KUKA KRL program: MyProgram_142().src

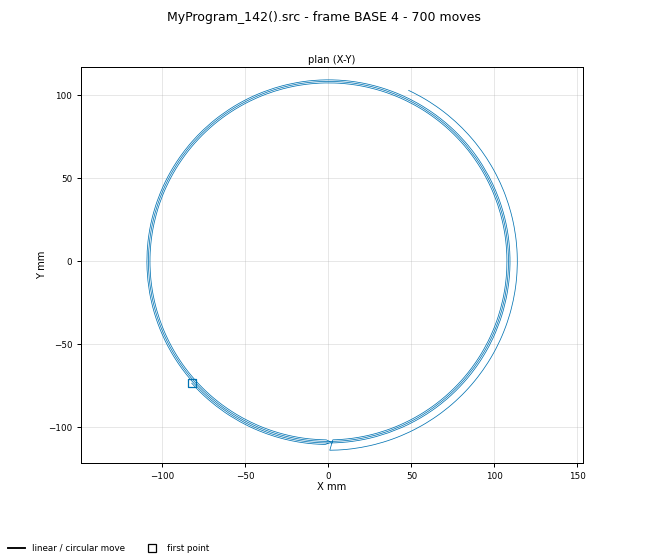
[picture p0: tool path of MyProgram_142().src in frame BASE 4, 700 of 700 moves have a stored position in this frame; points joined in program order, loops and branches not executed]
&ACCESS RVP
&REL 1
&PARAM TEMPLATE = C:\KRC\Roboter\Template\vorgabe
&PARAM EDITMASK = *
DEF MyProgram_142()
; ---- Setting reference (Base) ----
$BASE = BASE_DATA[4]

; --------------------------
; ---- Setting tool (TCP) ----
$TOOL = TOOL_DATA[3]
; --------------------------

$VEL.CP = VEL_APROX_PRINT
Startdeposition()
$VEL.CP = VEL_PRINT
LIN {X -82.3779,Y -73.3835,Z 113,A -141.7997,B 24.948,C -1.666,E1 24.8814,E2 227.604} C_DIS
LIN {X -79.9682,Y -76.004,Z 113,A -139.8537,B 24.948,C -1.6658,E1 24.8851,E2 225.6502} C_DIS
LIN {X -77.4714,Y -78.5454,Z 113,A -138.0878,B 24.9485,C -1.6585,E1 24.8886,E2 223.8941} C_DIS
LIN {X -74.7071,Y -81.1792,Z 113,A -136.1303,B 24.9488,C -1.6534,E1 24.8926,E2 221.9407} C_DIS
LIN {X -72.2466,Y -83.3774,Z 113,A -134.4348,B 24.949,C -1.6493,E1 24.8961,E2 220.2482} C_DIS
LIN {X -67.7785,Y -87.0492,Z 113,A -131.5023,B 24.9496,C -1.6408,E1 24.9025,E2 217.3249} C_DIS
LIN {X -62.2347,Y -91.0947,Z 113,A -127.8013,B 24.9496,C -1.6401,E1 24.9109,E2 213.6125} C_DIS
LIN {X -59.665,Y -92.797,Z 113,A -126.1786,B 24.9496,C -1.6385,E1 24.9147,E2 211.9885} C_DIS
LIN {X -53.2647,Y -96.6148,Z 113,A -122.4009,B 24.9503,C -1.6291,E1 24.9238,E2 208.2219} C_DIS
LIN {X -48.2181,Y -99.2292,Z 113,A -119.3028,B 24.9501,C -1.6312,E1 24.9315,E2 205.1103} C_DIS
LIN {X -45.3422,Y -100.5747,Z 113,A -117.6884,B 24.9503,C -1.628,E1 24.9356,E2 203.4997} C_DIS
LIN {X -41.9036,Y -102.0558,Z 113,A -114.9603,B 24.9485,C -1.6583,E1 24.9428,E2 200.6934} C_DIS
LIN {X -37.221,Y -103.8565,Z 113,A -113.2244,B 24.9508,C -1.6199,E1 24.9472,E2 199.0451} C_DIS
LIN {X -32.1983,Y -105.5211,Z 113,A -110.4618,B 24.9509,C -1.6183,E1 24.9545,E2 196.2811} C_DIS
LIN {X -28.3976,Y -106.6063,Z 113,A -108.4229,B 24.951,C -1.6164,E1 24.96,E2 194.2436} C_DIS
LIN {X -25.5467,Y -107.3263,Z 113,A -106.6947,B 24.9506,C -1.6239,E1 24.9647,E2 192.4952} C_DIS
LIN {X -22.1899,Y -108.0685,Z 113,A -105.0015,B 24.9509,C -1.6193,E1 24.9693,E2 190.8109} C_DIS
LIN {X -18.5186,Y -108.7583,Z 113,A -103.0189,B 24.9508,C -1.6204,E1 24.9748,E2 188.8237} C_DIS
LIN {X -15.3474,Y -109.2505,Z 113,A -101.4417,B 24.9511,C -1.6163,E1 24.9791,E2 187.255} C_DIS
LIN {X -12.6157,Y -109.5996,Z 113,A -100.0275,B 24.9511,C -1.6154,E1 24.983,E2 185.842} C_DIS
LIN {X -9.065,Y -109.9504,Z 113,A -98.0828,B 24.9509,C -1.6191,E1 24.9885,E2 183.8875} C_DIS
LIN {X -5.9741,Y -110.1613,Z 113,A -96.2315,B 24.9503,C -1.6294,E1 24.9937,E2 182.0111} C_DIS
LIN {X -2.0472,Y -110.3041,Z 113,A -94.0279,B 24.9498,C -1.6367,E1 24.9999,E2 179.7901} C_DIS
LIN {X -2.0472,Y -110.3041,Z 113,A -94.0279,B 24.9498,C -1.6367,E1 24.9999,E2 179.7901} C_DIS
Enddeposition()
LIN {X 0.8012,Y -109.3921,Z 113,A -93.8534,B 24.9521,C -1.5983,E1 25.0001,E2 179.7065} C_DIS
Startdeposition()
$VEL.CP = VEL_PRINT
LIN {X -2.7654,Y -109.365,Z 113,A -95.8153,B 24.9524,C -1.594,E1 24.9946,E2 181.6787} C_DIS
LIN {X -5.7929,Y -109.2451,Z 113,A -97.2879,B 24.9521,C -1.5986,E1 24.9905,E2 183.1408} C_DIS
LIN {X -8.9901,Y -109.0286,Z 113,A -98.9104,B 24.952,C -1.6009,E1 24.986,E2 184.7585} C_DIS
LIN {X -12.5666,Y -108.6743,Z 113,A -100.7989,B 24.952,C -1.6009,E1 24.9808,E2 186.6482} C_DIS
LIN {X -15.9909,Y -108.225,Z 113,A -102.74,B 24.9523,C -1.5959,E1 24.9754,E2 188.6028} C_DIS
LIN {X -19.4535,Y -107.6548,Z 113,A -104.4859,B 24.952,C -1.6002,E1 24.9706,E2 190.34} C_DIS
LIN {X -23.1089,Y -106.93,Z 113,A -106.4558,B 24.952,C -1.6003,E1 24.9652,E2 192.312} C_DIS
LIN {X -26.9087,Y -106.0378,Z 113,A -108.7166,B 24.9525,C -1.5927,E1 24.959,E2 194.594} C_DIS
LIN {X -30.6646,Y -105.0138,Z 113,A -110.6107,B 24.952,C -1.5999,E1 24.954,E2 196.4742} C_DIS
LIN {X -34.0937,Y -103.9509,Z 113,A -112.4944,B 24.952,C -1.6012,E1 24.949,E2 198.3582} C_DIS
LIN {X -37.5371,Y -102.7568,Z 113,A -114.8721,B 24.953,C -1.5842,E1 24.9426,E2 200.7808} C_DIS
LIN {X -41.2912,Y -101.3066,Z 113,A -116.4083,B 24.9515,C -1.609,E1 24.9388,E2 202.2615} C_DIS
LIN {X -44.4783,Y -99.9497,Z 113,A -118.2925,B 24.9515,C -1.6082,E1 24.9339,E2 204.1522} C_DIS
LIN {X -47.5492,Y -98.5246,Z 113,A -120.5665,B 24.9526,C -1.5905,E1 24.9281,E2 206.474} C_DIS
LIN {X -51.0831,Y -96.7395,Z 113,A -122.1173,B 24.9512,C -1.6138,E1 24.9244,E2 207.9737} C_DIS
LIN {X -56.8602,Y -93.4607,Z 113,A -125.5555,B 24.9508,C -1.6203,E1 24.9161,E2 211.4066} C_DIS
LIN {X -59.8344,Y -91.5863,Z 113,A -127.5128,B 24.9509,C -1.6186,E1 24.9114,E2 213.3743} C_DIS
LIN {X -66.1199,Y -87.1574,Z 113,A -131.2341,B 24.9498,C -1.6374,E1 24.9031,E2 217.0638} C_DIS
LIN {X -70.5458,Y -83.6155,Z 113,A -134.473,B 24.9501,C -1.6324,E1 24.896,E2 220.3268} C_DIS
LIN {X -73.0132,Y -81.4682,Z 113,A -136.1362,B 24.9497,C -1.6377,E1 24.8925,E2 221.9839} C_DIS
LIN {X -75.4532,Y -79.2163,Z 113,A -138.0378,B 24.9499,C -1.635,E1 24.8886,E2 223.8999} C_DIS
LIN {X -78.1128,Y -76.5934,Z 113,A -139.9944,B 24.9497,C -1.6392,E1 24.8847,E2 225.8547} C_DIS
LIN {X -80.6821,Y -73.881,Z 113,A -141.8513,B 24.9491,C -1.6474,E1 24.8812,E2 227.7003} C_DIS
LIN {X -83.2227,Y -71.0069,Z 113,A -143.8483,B 24.9488,C -1.6524,E1 24.8776,E2 229.6943} C_DIS
LIN {X -85.4937,Y -68.2577,Z 113,A -146.364,B 24.9501,C -1.6322,E1 24.8731,E2 232.27} C_DIS
LIN {X -88.0377,Y -64.9423,Z 113,A -147.7396,B 24.9478,C -1.6685,E1 24.8709,E2 233.5656} C_DIS
LIN {X -90.3611,Y -61.6687,Z 113,A -150.7884,B 24.9497,C -1.6379,E1 24.8659,E2 236.7024} C_DIS
LIN {X -92.8964,Y -57.7779,Z 113,A -152.5487,B 24.9478,C -1.6697,E1 24.8634,E2 238.3959} C_DIS
LIN {X -94.8352,Y -54.537,Z 113,A -154.5071,B 24.9474,C -1.6757,E1 24.8606,E2 240.3501} C_DIS
LIN {X -96.8538,Y -50.866,Z 113,A -156.705,B 24.947,C -1.6816,E1 24.8577,E2 242.5456} C_DIS
LIN {X -98.4649,Y -47.6735,Z 113,A -158.9102,B 24.9475,C -1.6743,E1 24.855,E2 244.78} C_DIS
LIN {X -100.2359,Y -43.8267,Z 113,A -160.6867,B 24.946,C -1.6973,E1 24.853,E2 246.5114} C_DIS
LIN {X -101.4514,Y -40.9354,Z 113,A -162.571,B 24.9463,C -1.693,E1 24.8509,E2 248.4166} C_DIS
LIN {X -102.8244,Y -37.3518,Z 113,A -164.4547,B 24.9456,C -1.7037,E1 24.8491,E2 250.2853} C_DIS
LIN {X -103.9435,Y -34.1167,Z 113,A -166.3425,B 24.9455,C -1.7055,E1 24.8474,E2 252.1797} C_DIS
LIN {X -104.9287,Y -30.9513,Z 113,A -168.2477,B 24.9455,C -1.7044,E1 24.8459,E2 254.0983} C_DIS
LIN {X -105.9399,Y -27.2899,Z 113,A -171.007,B 24.947,C -1.682,E1 24.8439,E2 256.9271} C_DIS
LIN {X -107.201,Y -21.8168,Z 113,A -173.3913,B 24.9451,C -1.7118,E1 24.8426,E2 259.2546} C_DIS
LIN {X -107.798,Y -18.6455,Z 113,A -174.9108,B 24.9443,C -1.7235,E1 24.8419,E2 260.7552} C_DIS
LIN {X -108.7762,Y -11.6534,Z 113,A -178.1709,B 24.9425,C -1.7516,E1 24.8407,E2 263.9678} C_DIS
LIN {X -109.2836,Y -5.0185,Z 113,A 177.3593,B 24.9442,C -1.7262,E1 24.8399,E2 268.5249} C_DIS
LIN {X -109.3981,Y -0.4851,Z 113,A 175.7323,B 24.9418,C -1.7616,E1 24.8398,E2 270.0774} C_DIS
LIN {X -109.2223,Y 6.206,Z 113,A 172.596,B 24.9402,C -1.7867,E1 24.8401,E2 273.1726} C_DIS
LIN {X -108.7527,Y 11.8781,Z 113,A 169.2354,B 24.9405,C -1.7821,E1 24.8408,E2 276.5644} C_DIS
LIN {X -108.4114,Y 14.675,Z 113,A 167.2505,B 24.9414,C -1.768,E1 24.8416,E2 278.5949} C_DIS
LIN {X -107.7858,Y 18.7251,Z 113,A 165.3486,B 24.9404,C -1.7839,E1 24.8424,E2 280.47} C_DIS
LIN {X -107.0836,Y 22.3884,Z 113,A 163.4098,B 24.9399,C -1.7908,E1 24.8435,E2 282.4039} C_DIS
LIN {X -106.2775,Y 25.9441,Z 113,A 161.1299,B 24.9404,C -1.7832,E1 24.845,E2 284.7153} C_DIS
LIN {X -105.3682,Y 29.423,Z 113,A 159.647,B 24.939,C -1.804,E1 24.8461,E2 286.1573} C_DIS
LIN {X -104.0831,Y 33.6853,Z 113,A 157.5878,B 24.9378,C -1.8215,E1 24.8477,E2 288.1865} C_DIS
LIN {X -103.2279,Y 36.2213,Z 113,A 155.9172,B 24.9382,C -1.8158,E1 24.8493,E2 289.8801} C_DIS
LIN {X -101.2858,Y 41.3425,Z 113,A 152.8339,B 24.9382,C -1.8167,E1 24.8524,E2 292.9786} C_DIS
LIN {X -99.7186,Y 44.9911,Z 113,A 150.9412,B 24.9372,C -1.83,E1 24.8545,E2 294.85} C_DIS
LIN {X -98.064,Y 48.4919,Z 113,A 148.8956,B 24.9369,C -1.8354,E1 24.857,E2 296.8937} C_DIS
LIN {X -96.7392,Y 51.0837,Z 113,A 147.4208,B 24.9364,C -1.8418,E1 24.8589,E2 298.3612} C_DIS
LIN {X -95.0536,Y 54.1568,Z 113,A 145.4662,B 24.9364,C -1.8427,E1 24.8616,E2 300.3239} C_DIS
LIN {X -93.3567,Y 57.0314,Z 113,A 143.353,B 24.9369,C -1.8342,E1 24.8647,E2 302.4684} C_DIS
LIN {X -91.542,Y 59.9015,Z 113,A 141.9274,B 24.9357,C -1.8523,E1 24.8668,E2 303.8578} C_DIS
LIN {X -89.57,Y 62.8125,Z 113,A 140.1452,B 24.9352,C -1.8597,E1 24.8696,E2 305.6313} C_DIS
LIN {X -86.8006,Y 66.586,Z 113,A 136.9244,B 24.9367,C -1.8376,E1 24.8751,E2 308.9202} C_DIS
LIN {X -83.8364,Y 70.2828,Z 113,A 135.274,B 24.9341,C -1.8752,E1 24.8779,E2 310.4886} C_DIS
LIN {X -82.098,Y 72.3057,Z 113,A 133.0171,B 24.9361,C -1.8465,E1 24.8822,E2 312.824} C_DIS
LIN {X -78.9179,Y 75.7628,Z 113,A 131.4131,B 24.9334,C -1.8848,E1 24.8851,E2 314.3437} C_DIS
LIN {X -75.4082,Y 79.259,Z 113,A 128.5636,B 24.9336,C -1.8814,E1 24.8909,E2 317.2134} C_DIS
LIN {X -70.6677,Y 83.5117,Z 113,A 125.2283,B 24.9331,C -1.889,E1 24.8978,E2 320.5437} C_DIS
LIN {X -68.3733,Y 85.4021,Z 113,A 123.6376,B 24.933,C -1.8911,E1 24.9013,E2 322.1353} C_DIS
LIN {X -65.5348,Y 87.5969,Z 113,A 121.7948,B 24.9326,C -1.8965,E1 24.9054,E2 323.9719} C_DIS
LIN {X -59.7976,Y 91.6105,Z 113,A 118.3589,B 24.9314,C -1.9127,E1 24.9132,E2 327.381} C_DIS
LIN {X -56.3625,Y 93.7632,Z 113,A 115.9531,B 24.9319,C -1.9058,E1 24.919,E2 329.8108} C_DIS
LIN {X -53.3037,Y 95.5338,Z 113,A 114.2429,B 24.9313,C -1.9145,E1 24.9231,E2 331.5052} C_DIS
LIN {X -50.6765,Y 96.9536,Z 113,A 112.6453,B 24.9312,C -1.9158,E1 24.927,E2 333.1041} C_DIS
LIN {X -48.0598,Y 98.2781,Z 113,A 111.1708,B 24.9308,C -1.9207,E1 24.9307,E2 334.571} C_DIS
LIN {X -45.59,Y 99.4482,Z 113,A 109.2316,B 24.9321,C -1.9032,E1 24.9357,E2 336.5565} C_DIS
LIN {X -42.5907,Y 100.7672,Z 113,A 107.9423,B 24.9307,C -1.9223,E1 24.9389,E2 337.8036} C_DIS
LIN {X -39.2401,Y 102.12,Z 113,A 105.8965,B 24.931,C -1.9189,E1 24.9443,E2 339.8618} C_DIS
LIN {X -32.8544,Y 104.3495,Z 113,A 102.6449,B 24.9298,C -1.9346,E1 24.9528,E2 343.0822} C_DIS
LIN {X -28.269,Y 105.6832,Z 113,A 99.7023,B 24.9309,C -1.9199,E1 24.9608,E2 346.0644} C_DIS
LIN {X -24.7509,Y 106.5617,Z 113,A 97.9468,B 24.9304,C -1.9274,E1 24.9655,E2 347.8046} C_DIS
LIN {X -18.6417,Y 107.8,Z 113,A 94.901,B 24.9295,C -1.9386,E1 24.9738,E2 350.827} C_DIS
LIN {X -15.5709,Y 108.2847,Z 113,A 93.1885,B 24.9297,C -1.9364,E1 24.9786,E2 352.5462} C_DIS
LIN {X -12.4417,Y 108.6889,Z 113,A 91.4662,B 24.9298,C -1.9346,E1 24.9833,E2 354.274} C_DIS
LIN {X -8.7221,Y 109.0501,Z 113,A 89.5604,B 24.9296,C -1.9376,E1 24.9886,E2 356.1736} C_DIS
LIN {X -5.0583,Y 109.2819,Z 113,A 87.5717,B 24.9298,C -1.9357,E1 24.9942,E2 358.1675} C_DIS
LIN {X -1.3425,Y 109.3921,Z 113,A 85.5642,B 24.9298,C -1.9337,E1 24.9998,E2 360.1797} C_DIS
LIN {X 2.3062,Y 109.3744,Z 113,A 83.6652,B 24.9298,C -1.9345,E1 25.0051,E2 362.0767} C_DIS
LIN {X 6.1411,Y 109.2259,Z 113,A 81.768,B 24.9295,C -1.9392,E1 25.0104,E2 363.9623} C_DIS
LIN {X 9.6682,Y 108.9709,Z 113,A 79.8747,B 24.9296,C -1.9374,E1 25.0156,E2 365.8589} C_DIS
LIN {X 13.002,Y 108.6233,Z 113,A 78.0458,B 24.9299,C -1.9341,E1 25.0207,E2 367.6942} C_DIS
LIN {X 16.8027,Y 108.1003,Z 113,A 76.1369,B 24.9296,C -1.9377,E1 25.026,E2 369.5929} C_DIS
LIN {X 20.5395,Y 107.453,Z 113,A 74.1322,B 24.9297,C -1.9361,E1 25.0315,E2 371.599} C_DIS
LIN {X 23.9831,Y 106.7391,Z 113,A 72.0822,B 24.9304,C -1.9267,E1 25.0371,E2 373.6687} C_DIS
LIN {X 27.6095,Y 105.8577,Z 113,A 70.3461,B 24.9298,C -1.9345,E1 25.0418,E2 375.3838} C_DIS
LIN {X 31.3079,Y 104.8229,Z 113,A 68.3615,B 24.9298,C -1.9342,E1 25.0471,E2 377.3658} C_DIS
LIN {X 34.8354,Y 103.7039,Z 113,A 65.8741,B 24.9316,C -1.91,E1 25.0538,E2 379.9057} C_DIS
LIN {X 38.5632,Y 102.3763,Z 113,A 64.6554,B 24.9292,C -1.9433,E1 25.0568,E2 381.0429} C_DIS
LIN {X 41.0421,Y 101.408,Z 113,A 62.9101,B 24.9304,C -1.9273,E1 25.0614,E2 382.8222} C_DIS
LIN {X 44.3336,Y 100.0149,Z 113,A 60.2503,B 24.9329,C -1.8925,E1 25.0684,E2 385.5578} C_DIS
LIN {X 48.9923,Y 97.8159,Z 113,A 58.6274,B 24.9299,C -1.9339,E1 25.0723,E2 387.0785} C_DIS
LIN {X 53.6545,Y 95.3379,Z 113,A 55.7155,B 24.9306,C -1.9239,E1 25.0795,E2 390.0056} C_DIS
LIN {X 56.3723,Y 93.7573,Z 113,A 53.9616,B 24.9311,C -1.9169,E1 25.0837,E2 391.7707} C_DIS
LIN {X 61.0705,Y 90.7656,Z 113,A 50.9637,B 24.9317,C -1.9089,E1 25.0907,E2 394.7777} C_DIS
LIN {X 64.5108,Y 88.3536,Z 113,A 48.6141,B 24.9324,C -1.8988,E1 25.0961,E2 397.143} C_DIS
LIN {X 67.3887,Y 86.1805,Z 113,A 46.9399,B 24.932,C -1.9044,E1 25.0998,E2 398.7978} C_DIS
LIN {X 70.6273,Y 83.5461,Z 113,A 44.7937,B 24.9322,C -1.9019,E1 25.1044,E2 400.9416} C_DIS
LIN {X 73.3173,Y 81.196,Z 113,A 42.8702,B 24.9326,C -1.8959,E1 25.1084,E2 402.8716} C_DIS
LIN {X 75.9181,Y 78.7683,Z 113,A 41.143,B 24.9325,C -1.8979,E1 25.1119,E2 404.5871} C_DIS
LIN {X 78.3464,Y 76.3557,Z 113,A 39.2407,B 24.9331,C -1.8893,E1 25.1156,E2 406.5017} C_DIS
LIN {X 81.9844,Y 72.4358,Z 113,A 36.4618,B 24.9335,C -1.8839,E1 25.1209,E2 409.281} C_DIS
LIN {X 84.1987,Y 69.8468,Z 113,A 33.9749,B 24.9359,C -1.8496,E1 25.1254,E2 411.8374} C_DIS
LIN {X 87.3366,Y 65.8814,Z 113,A 32.1429,B 24.9339,C -1.8782,E1 25.1284,E2 413.5934} C_DIS
LIN {X 89.3104,Y 63.181,Z 113,A 30.4798,B 24.9339,C -1.8776,E1 25.1311,E2 415.2498} C_DIS
LIN {X 90.9002,Y 60.8724,Z 113,A 28.8268,B 24.9347,C -1.8658,E1 25.1337,E2 416.9224} C_DIS
LIN {X 92.8626,Y 57.8322,Z 113,A 27.0985,B 24.9346,C -1.8681,E1 25.1363,E2 418.6366} C_DIS
LIN {X 96.5968,Y 51.3539,Z 113,A 23.357,B 24.9348,C -1.865,E1 25.1415,E2 422.366} C_DIS
LIN {X 98.9562,Y 46.647,Z 113,A 20.5663,B 24.9354,C -1.8557,E1 25.1449,E2 425.1635} C_DIS
LIN {X 100.73,Y 42.6791,Z 113,A 18.1538,B 24.9363,C -1.8432,E1 25.1476,E2 427.5925} C_DIS
LIN {X 102.7796,Y 37.4746,Z 113,A 15.2834,B 24.9367,C -1.8372,E1 25.1505,E2 430.4612} C_DIS
LIN {X 103.9222,Y 34.1824,Z 113,A 13.0549,B 24.9383,C -1.814,E1 25.1525,E2 432.7318} C_DIS
LIN {X 105.387,Y 29.3564,Z 113,A 10.8974,B 24.9374,C -1.8271,E1 25.1542,E2 434.8459} C_DIS
LIN {X 106.1589,Y 26.4299,Z 113,A 9.388,B 24.9375,C -1.8256,E1 25.1552,E2 436.3503} C_DIS
LIN {X 107.0513,Y 22.5459,Z 113,A 7.1063,B 24.9386,C -1.8105,E1 25.1566,E2 438.6544} C_DIS
LIN {X 107.6865,Y 19.2774,Z 113,A 5.4791,B 24.9386,C -1.8102,E1 25.1575,E2 440.2728} C_DIS
LIN {X 108.2497,Y 15.8174,Z 113,A 3.5533,B 24.9392,C -1.8004,E1 25.1583,E2 442.2104} C_DIS
LIN {X 108.6843,Y 12.4812,Z 113,A 1.921,B 24.9392,C -1.8004,E1 25.1589,E2 443.8328} C_DIS
LIN {X 109.0274,Y 9.0051,Z 113,A 0.011,B 24.9399,C -1.791,E1 25.1593,E2 445.7538} C_DIS
LIN {X 109.2436,Y 5.8206,Z 113,A -1.5956,B 24.94,C -1.7885,E1 25.1596,E2 447.3568} C_DIS
LIN {X 109.3762,Y 2.2106,Z 113,A -3.4948,B 24.9405,C -1.7821,E1 25.1598,E2 449.2599} C_DIS
LIN {X 109.3898,Y -1.4676,Z 113,A -5.4893,B 24.9411,C -1.7728,E1 25.1598,E2 451.2644} C_DIS
LIN {X 109.2818,Y -5.0597,Z 113,A -7.3747,B 24.9415,C -1.7665,E1 25.1595,E2 453.1534} C_DIS
LIN {X 108.9967,Y -9.3887,Z 113,A -9.5794,B 24.9418,C -1.7621,E1 25.1591,E2 455.3553} C_DIS
LIN {X 108.6501,Y -12.7727,Z 113,A -11.3391,B 24.9421,C -1.7573,E1 25.1585,E2 457.116} C_DIS
LIN {X 107.9142,Y -17.9587,Z 113,A -14.335,B 24.9434,C -1.7372,E1 25.1573,E2 460.1415} C_DIS
LIN {X 107.1046,Y -22.2864,Z 113,A -16.4,B 24.9432,C -1.7404,E1 25.1562,E2 462.1869} C_DIS
LIN {X 105.4172,Y -29.25,Z 113,A -20.4889,B 24.945,C -1.7136,E1 25.1533,E2 466.3156} C_DIS
LIN {X 104.4469,Y -32.5402,Z 113,A -21.8282,B 24.944,C -1.7281,E1 25.1522,E2 467.6131} C_DIS
LIN {X 103.4702,Y -35.5285,Z 113,A -23.5764,B 24.9447,C -1.7184,E1 25.1507,E2 469.3743} C_DIS
LIN {X 100.7111,Y -42.724,Z 113,A -27.546,B 24.9453,C -1.7088,E1 25.1466,E2 473.3445} C_DIS
LIN {X 99.1808,Y -46.1645,Z 113,A -29.4574,B 24.9455,C -1.7055,E1 25.1444,E2 475.2534} C_DIS
LIN {X 96.7449,Y -51.0728,Z 113,A -32.3463,B 24.9461,C -1.696,E1 25.1408,E2 478.1492} C_DIS
LIN {X 94.812,Y -54.5773,Z 113,A -35.0169,B 24.9481,C -1.6647,E1 25.137,E2 480.8799} C_DIS
LIN {X 92.529,Y -58.3655,Z 113,A -36.5246,B 24.9463,C -1.6934,E1 25.1349,E2 482.312} C_DIS
LIN {X 91.2221,Y -60.3867,Z 113,A -38.4148,B 24.9482,C -1.6623,E1 25.1319,E2 484.2664} C_DIS
LIN {X 89.1168,Y -63.4523,Z 113,A -39.8571,B 24.9472,C -1.679,E1 25.1296,E2 485.6622} C_DIS
LIN {X 86.3725,Y -67.1412,Z 113,A -42.8279,B 24.9491,C -1.6478,E1 25.1245,E2 488.6924} C_DIS
LIN {X 83.791,Y -70.3374,Z 113,A -44.4366,B 24.948,C -1.6658,E1 25.1217,E2 490.2513} C_DIS
LIN {X 81.4672,Y -73.0143,Z 113,A -46.2013,B 24.948,C -1.665,E1 25.1185,E2 492.01} C_DIS
LIN {X 79.0508,Y -75.6249,Z 113,A -48.1269,B 24.9485,C -1.6576,E1 25.1148,E2 493.9447} C_DIS
LIN {X 76.7151,Y -77.9925,Z 113,A -49.8185,B 24.9486,C -1.6555,E1 25.1114,E2 495.6341} C_DIS
LIN {X 73.9902,Y -80.5819,Z 113,A -51.7587,B 24.9489,C -1.652,E1 25.1075,E2 497.5744} C_DIS
LIN {X 71.3802,Y -82.9046,Z 113,A -53.8049,B 24.9497,C -1.6384,E1 25.1031,E2 499.6448} C_DIS
LIN {X 67.4867,Y -86.1016,Z 113,A -56.6817,B 24.9507,C -1.6223,E1 25.0968,E2 502.5488} C_DIS
LIN {X 64.6449,Y -88.2555,Z 113,A -57.9573,B 24.9494,C -1.6439,E1 25.094,E2 503.7688} C_DIS
LIN {X 62.2815,Y -89.9391,Z 113,A -60.1083,B 24.9512,C -1.6136,E1 25.089,E2 505.984} C_DIS
LIN {X 59.1447,Y -92.032,Z 113,A -61.6033,B 24.9502,C -1.6303,E1 25.0856,E2 507.4346} C_DIS
LIN {X 55.4697,Y -94.2929,Z 113,A -63.7913,B 24.9502,C -1.6292,E1 25.0804,E2 509.6185} C_DIS
LIN {X 52.2815,Y -96.0971,Z 113,A -66.5028,B 24.9525,C -1.592,E1 25.0735,E2 512.4101} C_DIS
LIN {X 47.8787,Y -98.3663,Z 113,A -68.1866,B 24.9504,C -1.6264,E1 25.0695,E2 514.008} C_DIS
LIN {X 44.4113,Y -99.9799,Z 113,A -70.5877,B 24.9517,C -1.6063,E1 25.0633,E2 516.4506} C_DIS
LIN {X 36.0671,Y -103.282,Z 113,A -74.9452,B 24.9512,C -1.6144,E1 25.052,E2 520.7795} C_DIS
LIN {X 28.6493,Y -105.5804,Z 113,A -79.1187,B 24.9517,C -1.6051,E1 25.0409,E2 524.9676} C_DIS
LIN {X 24.6705,Y -106.5803,Z 113,A -81.1297,B 24.9515,C -1.6088,E1 25.0354,E2 526.967} C_DIS
LIN {X 21.7324,Y -107.2183,Z 113,A -82.88,B 24.952,C -1.6,E1 25.0306,E2 528.7359} C_DIS
LIN {X 17.9909,Y -107.9089,Z 113,A -84.7608,B 24.9518,C -1.6031,E1 25.0254,E2 530.6072} C_DIS
LIN {X 14.2627,Y -108.4648,Z 113,A -86.7044,B 24.9518,C -1.6031,E1 25.0201,E2 532.5493} C_DIS
LIN {X 11.3431,Y -108.8087,Z 113,A -88.2669,B 24.952,C -1.6012,E1 25.0157,E2 534.1151} C_DIS
LIN {X 6.9829,Y -109.1759,Z 113,A -90.4253,B 24.9517,C -1.6056,E1 25.0097,E2 536.262} C_DIS
LIN {X 4.3324,Y -109.3131,Z 113,A -91.9065,B 24.952,C -1.6013,E1 25.0056,E2 537.7529} C_DIS
LIN {X 1.2624,Y -109.3926,Z 113,A -93.8285,B 24.9528,C -1.5878,E1 25.0001,E2 539.7065} C_DIS
LIN {X 1.2624,Y -109.3926,Z 113,A -93.8285,B 24.9528,C -1.5878,E1 25.0001,E2 539.7065} C_DIS
Enddeposition()
LIN {X 0.8016,Y -108.4705,Z 113,A -93.8436,B 24.9512,C -1.6134,E1 25.0003,E2 539.6609} C_DIS
Startdeposition()
$VEL.CP = VEL_PRINT
LIN {X 4.0415,Y -108.4,Z 113,A -91.1734,B 24.9488,C -1.6536,E1 25.008,E2 536.896} C_DIS
LIN {X 7.9739,Y -108.1818,Z 113,A -89.1291,B 24.9488,C -1.653,E1 25.0137,E2 534.854} C_DIS
LIN {X 11.5542,Y -107.8567,Z 113,A -87.3194,B 24.949,C -1.6503,E1 25.0187,E2 533.0518} C_DIS
LIN {X 15.2018,Y -107.403,Z 113,A -85.3984,B 24.949,C -1.6507,E1 25.024,E2 531.1314} C_DIS
LIN {X 18.8289,Y -106.8275,Z 113,A -83.4484,B 24.9488,C -1.6526,E1 25.0294,E2 529.1789} C_DIS
LIN {X 22.2338,Y -106.1713,Z 113,A -81.5918,B 24.9487,C -1.6553,E1 25.0345,E2 527.3183} C_DIS
LIN {X 28.4242,Y -104.6833,Z 113,A -78.3059,B 24.9487,C -1.6553,E1 25.0434,E2 524.037} C_DIS
LIN {X 34.797,Y -102.7409,Z 113,A -74.7828,B 24.9484,C -1.6597,E1 25.0528,E2 520.5101} C_DIS
LIN {X 37.9726,Y -101.6111,Z 113,A -72.9628,B 24.9481,C -1.6638,E1 25.0575,E2 518.6843} C_DIS
LIN {X 44.0864,Y -99.1119,Z 113,A -69.5353,B 24.948,C -1.6662,E1 25.0664,E2 515.2591} C_DIS
LIN {X 47.3058,Y -97.6155,Z 113,A -67.7699,B 24.948,C -1.6645,E1 25.0708,E2 513.5023} C_DIS
LIN {X 50.6503,Y -95.9222,Z 113,A -65.7577,B 24.9478,C -1.6692,E1 25.0758,E2 511.4845} C_DIS
LIN {X 53.5031,Y -94.3627,Z 113,A -63.8715,B 24.9471,C -1.6795,E1 25.0804,E2 509.5795} C_DIS
LIN {X 56.724,Y -92.4613,Z 113,A -61.8962,B 24.9469,C -1.6832,E1 25.0852,E2 507.6015} C_DIS
LIN {X 60.2765,Y -90.1868,Z 113,A -59.4491,B 24.946,C -1.6972,E1 25.0909,E2 505.1296} C_DIS
LIN {X 63.5812,Y -87.8882,Z 113,A -57.3098,B 24.9457,C -1.7021,E1 25.0958,E2 502.9861} C_DIS
LIN {X 68.1848,Y -84.3645,Z 113,A -54.0748,B 24.9448,C -1.7165,E1 25.1029,E2 499.7292} C_DIS
LIN {X 71.2151,Y -81.8227,Z 113,A -52.5492,B 24.9461,C -1.6965,E1 25.1061,E2 498.2568} C_DIS
LIN {X 73.8298,Y -79.4739,Z 113,A -50.5662,B 24.9454,C -1.7064,E1 25.1102,E2 496.2584} C_DIS
LIN {X 76.4474,Y -76.9571,Z 113,A -48.7093,B 24.9454,C -1.7084,E1 25.1139,E2 494.4045} C_DIS
LIN {X 78.986,Y -74.3486,Z 113,A -46.8645,B 24.9452,C -1.7098,E1 25.1174,E2 492.5644} C_DIS
LIN {X 81.4879,Y -71.5984,Z 113,A -44.8782,B 24.9448,C -1.7158,E1 25.1211,E2 490.5728} C_DIS
LIN {X 83.1038,Y -69.7175,Z 113,A -42.2227,B 24.9407,C -1.7793,E1 25.1261,E2 487.7798} C_DIS
LIN {X 87.7182,Y -63.8133,Z 113,A -39.6834,B 24.9441,C -1.7266,E1 25.1301,E2 485.3769} C_DIS
LIN {X 91.0597,Y -58.9475,Z 113,A -36.268,B 24.9427,C -1.7486,E1 25.1355,E2 481.9266} C_DIS
LIN {X 93.8673,Y -54.3653,Z 113,A -33.7392,B 24.9431,C -1.7431,E1 25.139,E2 479.4238} C_DIS
LIN {X 95.6402,Y -51.1843,Z 113,A -31.7471,B 24.9425,C -1.7518,E1 25.1417,E2 477.4215} C_DIS
LIN {X 97.6494,Y -47.2354,Z 113,A -29.5398,B 24.9425,C -1.7529,E1 25.1444,E2 475.2233} C_DIS
LIN {X 98.7831,Y -44.816,Z 113,A -28.2999,B 24.9426,C -1.7496,E1 25.1459,E2 473.9979} C_DIS
LIN {X 99.938,Y -42.1771,Z 113,A -26.2603,B 24.9408,C -1.7774,E1 25.1482,E2 471.904} C_DIS
LIN {X 101.1465,Y -39.1937,Z 113,A -24.8644,B 24.9413,C -1.7691,E1 25.1496,E2 470.5356} C_DIS
LIN {X 102.3599,Y -35.9019,Z 113,A -23.0977,B 24.9413,C -1.771,E1 25.1512,E2 468.7741} C_DIS
LIN {X 103.4178,Y -32.7362,Z 113,A -21.4254,B 24.9411,C -1.7725,E1 25.1527,E2 467.1077} C_DIS
LIN {X 104.4861,Y -29.1439,Z 113,A -19.3038,B 24.9403,C -1.7852,E1 25.1543,E2 464.9685} C_DIS
LIN {X 105.9416,Y -23.3005,Z 113,A -16.3319,B 24.9403,C -1.786,E1 25.1563,E2 462.0117} C_DIS
LIN {X 106.442,Y -20.899,Z 113,A -13.8196,B 24.9362,C -1.8448,E1 25.1577,E2 459.3755} C_DIS
LIN {X 107.477,Y -14.6811,Z 113,A -11.5165,B 24.9386,C -1.8094,E1 25.1585,E2 457.1695} C_DIS
LIN {X 107.9045,Y -11.0981,Z 113,A -9.7615,B 24.9386,C -1.8089,E1 25.1591,E2 455.4262} C_DIS
LIN {X 108.1829,Y -7.9607,Z 113,A -7.9698,B 24.9379,C -1.82,E1 25.1595,E2 453.6189} C_DIS
LIN {X 108.3918,Y -4.231,Z 113,A -6.004,B 24.9375,C -1.8261,E1 25.1597,E2 451.6503} C_DIS
LIN {X 108.4748,Y -0.1969,Z 113,A -3.8965,B 24.9371,C -1.8319,E1 25.1597,E2 449.5416} C_DIS
LIN {X 108.4184,Y 3.4591,Z 113,A -2.1075,B 24.9371,C -1.8319,E1 25.1597,E2 447.7634} C_DIS
LIN {X 108.24,Y 7.1169,Z 113,A -0.1588,B 24.9366,C -1.8387,E1 25.1594,E2 445.81} C_DIS
LIN {X 107.9555,Y 10.6079,Z 113,A 1.794,B 24.9359,C -1.8492,E1 25.1589,E2 443.8441} C_DIS
LIN {X 107.546,Y 14.1569,Z 113,A 3.5609,B 24.9359,C -1.8499,E1 25.1583,E2 442.086} C_DIS
LIN {X 107.0054,Y 17.7865,Z 113,A 5.5105,B 24.9354,C -1.8566,E1 25.1574,E2 440.1322} C_DIS
LIN {X 106.2965,Y 21.6237,Z 113,A 7.5317,B 24.9351,C -1.8613,E1 25.1563,E2 438.1117} C_DIS
LIN {X 105.5734,Y 24.9203,Z 113,A 9.1919,B 24.9351,C -1.8614,E1 25.1553,E2 436.4608} C_DIS
LIN {X 104.5831,Y 28.7951,Z 113,A 11.2922,B 24.9346,C -1.8674,E1 25.1538,E2 434.3585} C_DIS
LIN {X 103.1854,Y 33.4555,Z 113,A 13.9413,B 24.9338,C -1.8787,E1 25.1517,E2 431.6978} C_DIS
LIN {X 101.9982,Y 36.9182,Z 113,A 15.8722,B 24.9334,C -1.8843,E1 25.1499,E2 429.7645} C_DIS
LIN {X 100.5445,Y 40.7106,Z 113,A 18.0071,B 24.933,C -1.8902,E1 25.1477,E2 427.6276} C_DIS
LIN {X 99.143,Y 44.0175,Z 113,A 19.9124,B 24.9326,C -1.896,E1 25.1455,E2 425.7189} C_DIS
LIN {X 97.8899,Y 46.7349,Z 113,A 21.6723,B 24.9317,C -1.9084,E1 25.1434,E2 423.9392} C_DIS
LIN {X 96.0933,Y 50.3254,Z 113,A 23.5276,B 24.9321,C -1.9027,E1 25.1411,E2 422.1073} C_DIS
LIN {X 94.5124,Y 53.2359,Z 113,A 25.6811,B 24.9305,C -1.9252,E1 25.1381,E2 419.9118} C_DIS
LIN {X 92.8951,Y 56.0102,Z 113,A 27.0233,B 24.9313,C -1.9142,E1 25.1362,E2 418.6026} C_DIS
LIN {X 91.0066,Y 59.0303,Z 113,A 28.8362,B 24.9312,C -1.9162,E1 25.1335,E2 416.7942} C_DIS
LIN {X 88.7412,Y 62.384,Z 113,A 31.3085,B 24.9297,C -1.9362,E1 25.1295,E2 414.2866} C_DIS
LIN {X 83.2478,Y 69.5441,Z 113,A 35.8487,B 24.9296,C -1.9378,E1 25.1217,E2 409.764} C_DIS
LIN {X 80.8479,Y 72.3196,Z 113,A 37.7899,B 24.9293,C -1.9424,E1 25.1181,E2 407.8206} C_DIS
LIN {X 78.1175,Y 75.2606,Z 113,A 39.7514,B 24.9294,C -1.9403,E1 25.1144,E2 405.8727} C_DIS
LIN {X 75.5817,Y 77.808,Z 113,A 41.744,B 24.9288,C -1.9484,E1 25.1104,E2 403.8694} C_DIS
LIN {X 72.753,Y 80.4599,Z 113,A 43.7811,B 24.9286,C -1.9521,E1 25.1062,E2 401.8318} C_DIS
LIN {X 70.1707,Y 82.7202,Z 113,A 45.5669,B 24.9284,C -1.9545,E1 25.1024,E2 400.0472} C_DIS
LIN {X 67.3783,Y 85.0099,Z 113,A 47.4008,B 24.9284,C -1.9549,E1 25.0985,E2 398.2192} C_DIS
LIN {X 63.3687,Y 88.0404,Z 113,A 49.87,B 24.9286,C -1.9517,E1 25.093,E2 395.7665} C_DIS
LIN {X 57.1639,Y 92.1896,Z 113,A 53.9251,B 24.9278,C -1.9628,E1 25.0835,E2 391.6987} C_DIS
LIN {X 54.08,Y 94.0312,Z 113,A 55.8445,B 24.9275,C -1.9665,E1 25.0789,E2 389.7764} C_DIS
LIN {X 50.0566,Y 96.2349,Z 113,A 58.3558,B 24.927,C -1.9735,E1 25.0727,E2 387.2558} C_DIS
LIN {X 46.5453,Y 97.981,Z 113,A 60.6731,B 24.926,C -1.9864,E1 25.0668,E2 384.9139} C_DIS
LIN {X 42.5934,Y 99.7626,Z 113,A 62.7,B 24.9267,C -1.9779,E1 25.0617,E2 382.912} C_DIS
LIN {X 39.497,Y 101.0273,Z 113,A 64.4984,B 24.9264,C -1.981,E1 25.057,E2 381.1103} C_DIS
LIN {X 35.3462,Y 102.555,Z 113,A 66.8432,B 24.9262,C -1.9835,E1 25.0508,E2 378.7645} C_DIS
LIN {X 31.6672,Y 103.7493,Z 113,A 68.8553,B 24.9262,C -1.9838,E1 25.0455,E2 376.7552} C_DIS
LIN {X 29.187,Y 104.4738,Z 113,A 70.2663,B 24.926,C -1.9866,E1 25.0417,E2 375.3399} C_DIS
LIN {X 26.1077,Y 105.2856,Z 113,A 72.2782,B 24.9249,C -2.0013,E1 25.0361,E2 373.2961} C_DIS
LIN {X 22.589,Y 106.0968,Z 113,A 73.8135,B 24.926,C -1.9868,E1 25.032,E2 371.7972} C_DIS
LIN {X 18.7106,Y 106.8488,Z 113,A 75.8653,B 24.926,C -1.9862,E1 25.0264,E2 369.7491} C_DIS
LIN {X 15.2111,Y 107.4017,Z 113,A 77.7532,B 24.926,C -1.9875,E1 25.0212,E2 367.8601} C_DIS
LIN {X 11.4366,Y 107.869,Z 113,A 79.6768,B 24.9262,C -1.9843,E1 25.0159,E2 365.9453} C_DIS
LIN {X 8.3653,Y 108.1508,Z 113,A 81.4003,B 24.9259,C -1.9883,E1 25.0111,E2 364.2134} C_DIS
LIN {X 4.714,Y 108.3711,Z 113,A 83.2079,B 24.9263,C -1.9832,E1 25.0061,E2 362.4185} C_DIS
LIN {X 1.3208,Y 108.4674,Z 113,A 85.1608,B 24.9258,C -1.9894,E1 25.0006,E2 360.4511} C_DIS
LIN {X -2.2772,Y 108.45,Z 113,A 87.0206,B 24.926,C -1.9873,E1 24.9954,E2 358.5961} C_DIS
LIN {X -5.4799,Y 108.3362,Z 113,A 88.6814,B 24.926,C -1.9854,E1 24.9908,E2 356.9394} C_DIS
LIN {X -9.0105,Y 108.0993,Z 113,A 90.5596,B 24.9261,C -1.985,E1 24.9855,E2 355.0616} C_DIS
LIN {X -12.6757,Y 107.7304,Z 113,A 92.4542,B 24.9264,C -1.9819,E1 24.9803,E2 353.1731} C_DIS
LIN {X -16.0723,Y 107.2774,Z 113,A 94.2223,B 24.9266,C -1.979,E1 24.9754,E2 351.4105} C_DIS
LIN {X -19.16,Y 106.768,Z 113,A 96.6333,B 24.9244,C -2.0081,E1 24.9686,E2 348.9277} C_DIS
LIN {X -23.763,Y 105.8407,Z 113,A 98.5354,B 24.9263,C -1.9828,E1 24.9636,E2 347.0836} C_DIS
LIN {X -27.3044,Y 104.9813,Z 113,A 101.1843,B 24.9243,C -2.0098,E1 24.9562,E2 344.3666} C_DIS
LIN {X -32.2607,Y 103.5653,Z 113,A 103.0313,B 24.9271,C -1.9719,E1 24.9515,E2 342.6065} C_DIS
LIN {X -36.7532,Y 102.0583,Z 113,A 105.6198,B 24.9271,C -1.9721,E1 24.9447,E2 340.0125} C_DIS
LIN {X -39.853,Y 100.8875,Z 113,A 107.3861,B 24.9272,C -1.9704,E1 24.9401,E2 338.2466} C_DIS
LIN {X -43.45,Y 99.3912,Z 113,A 109.2935,B 24.9279,C -1.9615,E1 24.9352,E2 336.3558} C_DIS
LIN {X -46.5112,Y 97.9973,Z 113,A 111.1345,B 24.9279,C -1.9613,E1 24.9305,E2 334.5108} C_DIS
LIN {X -49.5708,Y 96.4847,Z 113,A 112.9928,B 24.9279,C -1.9605,E1 24.9259,E2 332.6493} C_DIS
LIN {X -52.8348,Y 94.7364,Z 113,A 114.9937,B 24.9281,C -1.9589,E1 24.921,E2 330.6466} C_DIS
LIN {X -56.2257,Y 92.7642,Z 113,A 117.0128,B 24.9285,C -1.9531,E1 24.9162,E2 328.6353} C_DIS
LIN {X -58.7616,Y 91.1791,Z 113,A 118.6213,B 24.9286,C -1.9512,E1 24.9124,E2 327.0261} C_DIS
LIN {X -62.5413,Y 88.6307,Z 113,A 121.1351,B 24.9286,C -1.9504,E1 24.9066,E2 324.5056} C_DIS
LIN {X -65.3973,Y 86.5436,Z 113,A 123.0045,B 24.929,C -1.9466,E1 24.9024,E2 322.6387} C_DIS
LIN {X -68.355,Y 84.2265,Z 113,A 124.9127,B 24.9295,C -1.9393,E1 24.8982,E2 320.7407} C_DIS
LIN {X -71.019,Y 81.9939,Z 113,A 126.9495,B 24.9292,C -1.9429,E1 24.8939,E2 318.6875} C_DIS
LIN {X -74.2997,Y 79.032,Z 113,A 129.1248,B 24.9301,C -1.9313,E1 24.8895,E2 316.5309} C_DIS
LIN {X -77.441,Y 75.9575,Z 113,A 131.6789,B 24.9298,C -1.9346,E1 24.8844,E2 313.9583} C_DIS
LIN {X -81.1167,Y 72.0193,Z 113,A 134.3397,B 24.9309,C -1.9203,E1 24.8794,E2 311.3196} C_DIS
LIN {X -83.3177,Y 69.46,Z 113,A 136.0766,B 24.9313,C -1.914,E1 24.8763,E2 309.59} C_DIS
LIN {X -85.0367,Y 67.3445,Z 113,A 137.7453,B 24.931,C -1.9188,E1 24.8734,E2 307.9018} C_DIS
LIN {X -87.9279,Y 63.5263,Z 113,A 140.1108,B 24.9319,C -1.9057,E1 24.8695,E2 305.5562} C_DIS
LIN {X -89.8465,Y 60.7792,Z 113,A 141.8152,B 24.9324,C -1.8983,E1 24.8668,E2 303.861} C_DIS
LIN {X -91.646,Y 58.0341,Z 113,A 143.7946,B 24.9321,C -1.9026,E1 24.8638,E2 301.8612} C_DIS
LIN {X -93.9101,Y 54.2907,Z 113,A 145.8232,B 24.9334,C -1.8854,E1 24.8609,E2 299.8634} C_DIS
LIN {X -95.2183,Y 51.9621,Z 113,A 147.4034,B 24.9332,C -1.8876,E1 24.8588,E2 298.2695} C_DIS
LIN {X -96.8798,Y 48.7963,Z 113,A 149.7803,B 24.9323,C -1.9004,E1 24.8557,E2 295.8493} C_DIS
LIN {X -98.5419,Y 45.3457,Z 113,A 151.7807,B 24.9328,C -1.8934,E1 24.8534,E2 293.8547} C_DIS
LIN {X -100.0042,Y 42.0199,Z 113,A 153.802,B 24.9329,C -1.8914,E1 24.8512,E2 291.8268} C_DIS
LIN {X -101.5089,Y 38.2424,Z 113,A 155.4479,B 24.9347,C -1.8658,E1 24.8496,E2 290.2327} C_DIS
LIN {X -102.7681,Y 34.7163,Z 113,A 157.3629,B 24.9353,C -1.8573,E1 24.8479,E2 288.3273} C_DIS
LIN {X -103.8564,Y 31.3143,Z 113,A 159.1848,B 24.9359,C -1.8489,E1 24.8463,E2 286.5148} C_DIS
LIN {X -104.5113,Y 29.0548,Z 113,A 160.6436,B 24.9356,C -1.8531,E1 24.8452,E2 285.0377} C_DIS
LIN {X -105.4242,Y 25.5396,Z 113,A 162.4855,B 24.9363,C -1.8441,E1 24.844,E2 283.2065} C_DIS
LIN {X -106.1277,Y 22.4462,Z 113,A 164.1843,B 24.9366,C -1.8396,E1 24.843,E2 281.5084} C_DIS
LIN {X -106.7509,Y 19.2549,Z 113,A 165.9647,B 24.9368,C -1.8364,E1 24.8421,E2 279.725} C_DIS
LIN {X -107.2629,Y 16.1661,Z 113,A 167.8674,B 24.9365,C -1.8404,E1 24.8413,E2 277.8015} C_DIS
LIN {X -107.7008,Y 12.928,Z 113,A 170.4068,B 24.9348,C -1.8657,E1 24.8404,E2 275.1865} C_DIS
LIN {X -108.2748,Y 6.5903,Z 113,A 173.1207,B 24.9372,C -1.8301,E1 24.8399,E2 272.5412} C_DIS
LIN {X -108.4283,Y 3.1391,Z 113,A 174.7901,B 24.938,C -1.8184,E1 24.8399,E2 270.8897} C_DIS
LIN {X -108.4693,Y -1.067,Z 113,A 176.9646,B 24.9386,C -1.8094,E1 24.8399,E2 268.7236} C_DIS
LIN {X -108.3488,Y -5.2324,Z 113,A 179.8941,B 24.9372,C -1.8298,E1 24.8403,E2 265.7276} C_DIS
LIN {X -107.941,Y -10.749,Z 113,A -178.2396,B 24.9406,C -1.7805,E1 24.8407,E2 263.9678} C_DIS
LIN {X -107.5063,Y -14.4509,Z 113,A -175.8992,B 24.9401,C -1.7882,E1 24.8415,E2 261.5949} C_DIS
LIN {X -106.4275,Y -20.9743,Z 113,A -172.523,B 24.9411,C -1.7728,E1 24.8431,E2 258.2356} C_DIS
LIN {X -105.7707,Y -24.0663,Z 113,A -170.6091,B 24.9408,C -1.7768,E1 24.8443,E2 256.3008} C_DIS
LIN {X -104.6521,Y -28.5398,Z 113,A -168.4022,B 24.9419,C -1.7607,E1 24.8459,E2 254.1195} C_DIS
LIN {X -103.6889,Y -31.8622,Z 113,A -166.8077,B 24.9428,C -1.7464,E1 24.8471,E2 252.55} C_DIS
LIN {X -102.9232,Y -34.2564,Z 113,A -165.1671,B 24.9423,C -1.7542,E1 24.8486,E2 250.8814} C_DIS
LIN {X -101.5457,Y -38.1452,Z 113,A -163.1072,B 24.9431,C -1.7432,E1 24.8505,E2 248.8361} C_DIS
LIN {X -100.5121,Y -40.7901,Z 113,A -161.3769,B 24.9428,C -1.7476,E1 24.8523,E2 247.0856} C_DIS
LIN {X -99.1591,Y -43.9817,Z 113,A -159.3615,B 24.9427,C -1.7493,E1 24.8546,E2 245.0551} C_DIS
LIN {X -97.2611,Y -48.0292,Z 113,A -157.354,B 24.944,C -1.7291,E1 24.857,E2 243.0847} C_DIS
LIN {X -95.5107,Y -51.4231,Z 113,A -155.3182,B 24.9443,C -1.7243,E1 24.8597,E2 241.0497} C_DIS
LIN {X -93.7571,Y -54.557,Z 113,A -153.4133,B 24.9446,C -1.7194,E1 24.8623,E2 239.1464} C_DIS
LIN {X -92.0169,Y -57.4404,Z 113,A -151.3653,B 24.9442,C -1.7251,E1 24.8653,E2 237.0744} C_DIS
LIN {X -89.5413,Y -61.2299,Z 113,A -149.3067,B 24.9454,C -1.7061,E1 24.8685,E2 235.0507} C_DIS
LIN {X -87.6493,Y -63.9073,Z 113,A -147.5082,B 24.9456,C -1.7044,E1 24.8714,E2 233.2476} C_DIS
LIN {X -85.8732,Y -66.2745,Z 113,A -145.6712,B 24.9451,C -1.7111,E1 24.8746,E2 231.3858} C_DIS
LIN {X -82.962,Y -69.8869,Z 113,A -143.3769,B 24.9459,C -1.6993,E1 24.8786,E2 229.1091} C_DIS
LIN {X -80.633,Y -72.5596,Z 113,A -141.5007,B 24.9461,C -1.6952,E1 24.8821,E2 227.2342} C_DIS
LIN {X -78.1243,Y -75.2536,Z 113,A -139.6564,B 24.9467,C -1.687,E1 24.8856,E2 225.4013} C_DIS
LIN {X -75.5932,Y -77.7969,Z 113,A -137.7085,B 24.9467,C -1.685,E1 24.8895,E2 223.45} C_DIS
LIN {X -73.1972,Y -80.0545,Z 113,A -135.9215,B 24.9469,C -1.6834,E1 24.8932,E2 221.6597} C_DIS
LIN {X -70.1455,Y -82.7417,Z 113,A -133.5189,B 24.9465,C -1.6892,E1 24.8983,E2 219.2338} C_DIS
LIN {X -66.2279,Y -85.9091,Z 113,A -131.1481,B 24.9476,C -1.6729,E1 24.9034,E2 216.893} C_DIS
LIN {X -63.2545,Y -88.1219,Z 113,A -128.7769,B 24.9467,C -1.6859,E1 24.9089,E2 214.4827} C_DIS
LIN {X -60.4833,Y -90.0468,Z 113,A -127.2911,B 24.9477,C -1.6712,E1 24.9122,E2 213.0268} C_DIS
LIN {X -57.9021,Y -91.7284,Z 113,A -125.6806,B 24.9479,C -1.668,E1 24.916,E2 211.4188} C_DIS
LIN {X -55.5194,Y -93.1893,Z 113,A -124.0678,B 24.9477,C -1.6713,E1 24.9199,E2 209.7932} C_DIS
LIN {X -51.901,Y -95.2514,Z 113,A -122.0112,B 24.9482,C -1.6625,E1 24.9249,E2 207.7515} C_DIS
LIN {X -48.9589,Y -96.7974,Z 113,A -120.1228,B 24.948,C -1.6656,E1 24.9296,E2 205.8508} C_DIS
LIN {X -45.0288,Y -98.6872,Z 113,A -117.9282,B 24.9485,C -1.6585,E1 24.9352,E2 203.6673} C_DIS
LIN {X -41.8786,Y -100.0638,Z 113,A -116.0882,B 24.9485,C -1.6576,E1 24.9399,E2 201.8254} C_DIS
LIN {X -37.8785,Y -101.6467,Z 113,A -113.8302,B 24.9487,C -1.6548,E1 24.9458,E2 199.5691} C_DIS
LIN {X -34.3132,Y -102.9041,Z 113,A -111.8519,B 24.9488,C -1.6524,E1 24.951,E2 197.5927} C_DIS
LIN {X -30.0147,Y -104.2393,Z 113,A -108.971,B 24.9477,C -1.6713,E1 24.9588,E2 194.6623} C_DIS
LIN {X -26.1735,Y -105.2696,Z 113,A -107.3974,B 24.9491,C -1.6485,E1 24.963,E2 193.1405} C_DIS
LIN {X -23.0995,Y -105.9855,Z 113,A -105.6739,B 24.949,C -1.65,E1 24.9677,E2 191.4111} C_DIS
LIN {X -19.1733,Y -106.7656,Z 113,A -103.6282,B 24.9492,C -1.6464,E1 24.9733,E2 189.3718} C_DIS
LIN {X -15.4202,Y -107.372,Z 113,A -101.6432,B 24.9492,C -1.645,E1 24.9787,E2 187.3886} C_DIS
LIN {X -12.0401,Y -107.8048,Z 113,A -99.786,B 24.9492,C -1.647,E1 24.9839,E2 185.5253} C_DIS
LIN {X -8.9179,Y -108.1067,Z 113,A -98.1374,B 24.9492,C -1.6466,E1 24.9885,E2 183.8768} C_DIS
LIN {X -5.0124,Y -108.3582,Z 113,A -96.2196,B 24.9496,C -1.6405,E1 24.9938,E2 181.9729} C_DIS
LIN {X -2.0343,Y -108.4545,Z 113,A -94.6857,B 24.9496,C -1.6391,E1 24.9981,E2 180.4421} C_DIS
LIN {X 0.8016,Y -108.4705,Z 113,A -93.8414,B 24.9513,C -1.6125,E1 25.0003,E2 179.6609} C_DIS
Enddeposition()
LIN {X 0.8016,Y -108.4705,Z 113,A -93.8414,B 24.9513,C -1.6125,E1 25.0003,E2 179.6609} C_DIS
Startdeposition()
$VEL.CP = VEL_PRINT
LIN {X -1.3239,Y -107.5426,Z 113,A -94.916,B 24.9502,C -1.6309,E1 24.9974,E2 180.692} C_DIS
LIN {X -3.5841,Y -107.4894,Z 113,A -96.1655,B 24.9502,C -1.6289,E1 24.9939,E2 181.9463} C_DIS
LIN {X -6.2176,Y -107.3692,Z 113,A -97.5683,B 24.9502,C -1.6289,E1 24.99,E2 183.3495} C_DIS
LIN {X -8.8457,Y -107.1847,Z 113,A -98.9716,B 24.9502,C -1.6289,E1 24.9861,E2 184.7534} C_DIS
LIN {X -11.4685,Y -106.9358,Z 113,A -100.5263,B 24.9506,C -1.623,E1 24.9817,E2 186.3229} C_DIS
LIN {X -15.1941,Y -106.4701,Z 113,A -102.3754,B 24.9502,C -1.6295,E1 24.9766,E2 188.1582} C_DIS
LIN {X -18.3888,Y -105.967,Z 113,A -104.0582,B 24.9502,C -1.6315,E1 24.972,E2 189.8376} C_DIS
LIN {X -21.8948,Y -105.2968,Z 113,A -105.9622,B 24.9501,C -1.6322,E1 24.9668,E2 191.7421} C_DIS
LIN {X -24.383,Y -104.7484,Z 113,A -107.4014,B 24.9502,C -1.6296,E1 24.9628,E2 193.1892} C_DIS
LIN {X -27.2386,Y -104.0434,Z 113,A -108.876,B 24.95,C -1.6342,E1 24.9589,E2 194.6552} C_DIS
LIN {X -29.9571,Y -103.2944,Z 113,A -110.3935,B 24.95,C -1.6346,E1 24.9548,E2 196.1742} C_DIS
LIN {X -33.3793,Y -102.2381,Z 113,A -112.3475,B 24.95,C -1.6342,E1 24.9496,E2 198.1325} C_DIS
LIN {X -35.8709,Y -101.3907,Z 113,A -113.7521,B 24.9499,C -1.6353,E1 24.9459,E2 199.5373} C_DIS
LIN {X -39.586,Y -99.9988,Z 113,A -115.871,B 24.9498,C -1.6371,E1 24.9403,E2 201.6564} C_DIS
LIN {X -42.3757,Y -98.8507,Z 113,A -117.4388,B 24.9496,C -1.6403,E1 24.9363,E2 203.2202} C_DIS
LIN {X -44.7858,Y -97.7824,Z 113,A -118.8471,B 24.9495,C -1.6417,E1 24.9327,E2 204.6286} C_DIS
LIN {X -46.8284,Y -96.8189,Z 113,A -120.1015,B 24.9495,C -1.6412,E1 24.9295,E2 205.8875} C_DIS
LIN {X -49.5385,Y -95.4625,Z 113,A -121.6684,B 24.9493,C -1.645,E1 24.9257,E2 207.4494} C_DIS
LIN {X -51.5218,Y -94.405,Z 113,A -122.9149,B 24.9493,C -1.6447,E1 24.9226,E2 208.7001} C_DIS
LIN {X -55.298,Y -92.2458,Z 113,A -125.1945,B 24.949,C -1.6495,E1 24.9171,E2 210.9751} C_DIS
LIN {X -58.3293,Y -90.3576,Z 113,A -127.15,B 24.949,C -1.6504,E1 24.9125,E2 212.9347} C_DIS
LIN {X -60.8694,Y -88.6682,Z 113,A -128.7234,B 24.9487,C -1.655,E1 24.9088,E2 214.5024} C_DIS
LIN {X -64.0742,Y -86.3809,Z 113,A -130.8396,B 24.9485,C -1.6579,E1 24.904,E2 216.6191} C_DIS
LIN {X -65.9422,Y -84.9617,Z 113,A -132.1987,B 24.9486,C -1.656,E1 24.901,E2 217.9877} C_DIS
LIN {X -68.7223,Y -82.7283,Z 113,A -134.0508,B 24.9483,C -1.6614,E1 24.897,E2 219.834} C_DIS
LIN {X -71.094,Y -80.7006,Z 113,A -135.8631,B 24.9484,C -1.6589,E1 24.8932,E2 221.6592} C_DIS
LIN {X -73.6854,Y -78.3402,Z 113,A -137.5909,B 24.9479,C -1.668,E1 24.8897,E2 223.3724} C_DIS
LIN {X -75.9156,Y -76.1825,Z 113,A -139.3949,B 24.948,C -1.6658,E1 24.886,E2 225.1894} C_DIS
LIN {X -78.3443,Y -73.6811,Z 113,A -141.1185,B 24.9474,C -1.6749,E1 24.8827,E2 226.8986} C_DIS
LIN {X -80.4374,Y -71.3917,Z 113,A -142.9205,B 24.9476,C -1.673,E1 24.8794,E2 228.7132} C_DIS
LIN {X -82.7083,Y -68.7464,Z 113,A -144.6179,B 24.9469,C -1.6833,E1 24.8763,E2 230.3937} C_DIS
LIN {X -84.3892,Y -66.6723,Z 113,A -146.1169,B 24.9469,C -1.6839,E1 24.8737,E2 231.8985} C_DIS
LIN {X -86.3911,Y -64.0603,Z 113,A -147.793,B 24.9464,C -1.691,E1 24.8709,E2 233.5656} C_DIS
LIN {X -87.9318,Y -61.9287,Z 113,A -149.2063,B 24.9462,C -1.6941,E1 24.8686,E2 234.9786} C_DIS
LIN {X -89.9335,Y -58.981,Z 113,A -151.1063,B 24.9459,C -1.6989,E1 24.8656,E2 236.8765} C_DIS
LIN {X -91.5638,Y -56.4201,Z 113,A -152.742,B 24.9457,C -1.7024,E1 24.8632,E2 238.5121} C_DIS
LIN {X -93.2546,Y -53.5753,Z 113,A -154.5692,B 24.9455,C -1.7048,E1 24.8606,E2 240.3431} C_DIS
LIN {X -94.8548,Y -50.6925,Z 113,A -156.2787,B 24.9451,C -1.7113,E1 24.8583,E2 242.0461} C_DIS
LIN {X -96.4824,Y -47.5178,Z 113,A -158.2366,B 24.9449,C -1.7145,E1 24.8559,E2 244.0068} C_DIS
LIN {X -98.17,Y -43.9257,Z 113,A -160.3206,B 24.9444,C -1.7217,E1 24.8534,E2 246.0852} C_DIS
LIN {X -99.2094,Y -41.5247,Z 113,A -161.7698,B 24.9444,C -1.7237,E1 24.8519,E2 247.5377} C_DIS
LIN {X -100.5352,Y -38.2024,Z 113,A -163.6957,B 24.944,C -1.7285,E1 24.8499,E2 249.4628} C_DIS
LIN {X -101.7018,Y -34.9842,Z 113,A -165.4756,B 24.9435,C -1.7355,E1 24.8482,E2 251.2361} C_DIS
LIN {X -102.5283,Y -32.4826,Z 113,A -166.8911,B 24.9433,C -1.7393,E1 24.847,E2 252.6506} C_DIS
LIN {X -103.2931,Y -29.9614,Z 113,A -168.3026,B 24.943,C -1.7433,E1 24.8459,E2 254.0609} C_DIS
LIN {X -103.9992,Y -27.4103,Z 113,A -169.7234,B 24.9428,C -1.7472,E1 24.8449,E2 255.4805} C_DIS
LIN {X -104.8545,Y -23.9238,Z 113,A -171.6908,B 24.9425,C -1.7512,E1 24.8436,E2 257.45} C_DIS
LIN {X -105.636,Y -20.1935,Z 113,A -173.7373,B 24.9421,C -1.757,E1 24.8425,E2 259.4948} C_DIS
LIN {X -106.1387,Y -17.3624,Z 113,A -175.2891,B 24.9419,C -1.761,E1 24.8417,E2 261.0461} C_DIS
LIN {X -106.5781,Y -14.43,Z 113,A -176.8187,B 24.9414,C -1.7679,E1 24.8411,E2 262.5686} C_DIS
LIN {X -106.9854,Y -10.9957,Z 113,A -178.692,B 24.9411,C -1.7727,E1 24.8405,E2 264.4417} C_DIS
LIN {X -107.2657,Y -7.8182,Z 113,A 179.653,B 24.9406,C -1.7797,E1 24.8402,E2 266.0898} C_DIS
LIN {X -107.4235,Y -5.2232,Z 113,A 178.2385,B 24.9404,C -1.7831,E1 24.8399,E2 267.5047} C_DIS
LIN {X -107.5188,Y -2.6134,Z 113,A 176.8237,B 24.9402,C -1.7867,E1 24.8399,E2 268.9194} C_DIS
LIN {X -107.5499,Y -0.2195,Z 113,A 175.4961,B 24.94,C -1.7889,E1 24.8398,E2 270.2497} C_DIS
LIN {X -107.5188,Y 2.6179,Z 113,A 174.0075,B 24.9396,C -1.7947,E1 24.8398,E2 271.7336} C_DIS
LIN {X -107.4203,Y 5.2942,Z 113,A 172.5756,B 24.9393,C -1.7991,E1 24.84,E2 273.1636} C_DIS
LIN {X -107.2538,Y 7.9815,Z 113,A 171.157,B 24.939,C -1.8043,E1 24.8403,E2 274.5782} C_DIS
LIN {X -107.0297,Y 10.572,Z 113,A 169.7426,B 24.9387,C -1.8078,E1 24.8407,E2 275.9929} C_DIS
LIN {X -106.6364,Y 13.9796,Z 113,A 167.8636,B 24.9385,C -1.8118,E1 24.8413,E2 277.8735} C_DIS
LIN {X -106.2404,Y 16.7273,Z 113,A 166.3528,B 24.9382,C -1.8155,E1 24.8419,E2 279.3846} C_DIS
LIN {X -105.7317,Y 19.6966,Z 113,A 164.7868,B 24.9378,C -1.822,E1 24.8427,E2 280.9442} C_DIS
LIN {X -105.0532,Y 23.0341,Z 113,A 162.8775,B 24.9376,C -1.8244,E1 24.8438,E2 282.8591} C_DIS
LIN {X -104.3297,Y 26.124,Z 113,A 161.2522,B 24.9371,C -1.8322,E1 24.8448,E2 284.4754} C_DIS
LIN {X -103.759,Y 28.2998,Z 113,A 160,B 24.9369,C -1.834,E1 24.8457,E2 285.7304} C_DIS
LIN {X -102.6443,Y 32.1083,Z 113,A 157.9153,B 24.9364,C -1.8418,E1 24.8474,E2 287.8087} C_DIS
LIN {X -101.7007,Y 34.9876,Z 113,A 156.2915,B 24.9361,C -1.8465,E1 24.8488,E2 289.4305} C_DIS
LIN {X -100.8131,Y 37.4683,Z 113,A 154.879,B 24.9358,C -1.8505,E1 24.8502,E2 290.8414} C_DIS
LIN {X -99.9732,Y 39.6512,Z 113,A 153.5737,B 24.9357,C -1.8522,E1 24.8515,E2 292.15} C_DIS
LIN {X -98.8969,Y 42.2661,Z 113,A 152.0943,B 24.9353,C -1.8578,E1 24.8531,E2 293.6243} C_DIS
LIN {X -97.7805,Y 44.7899,Z 113,A 150.6286,B 24.935,C -1.8624,E1 24.8548,E2 295.087} C_DIS
LIN {X -96.0638,Y 48.3621,Z 113,A 148.5032,B 24.9346,C -1.8682,E1 24.8574,E2 297.21} C_DIS
LIN {X -94.8505,Y 50.7006,Z 113,A 147.0902,B 24.9343,C -1.872,E1 24.8592,E2 298.6214} C_DIS
LIN {X -93.3892,Y 53.3411,Z 113,A 145.3841,B 24.9343,C -1.8732,E1 24.8616,E2 300.3339} C_DIS
LIN {X -91.7629,Y 56.0925,Z 113,A 143.7557,B 24.9337,C -1.8808,E1 24.8639,E2 301.9524} C_DIS
LIN {X -90.3526,Y 58.3371,Z 113,A 142.2936,B 24.9335,C -1.883,E1 24.8661,E2 303.4167} C_DIS
LIN {X -88.6833,Y 60.8476,Z 113,A 140.7226,B 24.9331,C -1.8887,E1 24.8685,E2 304.9819} C_DIS
LIN {X -86.3896,Y 64.0625,Z 113,A 138.5893,B 24.9328,C -1.8934,E1 24.872,E2 307.1144} C_DIS
LIN {X -84.4847,Y 66.5515,Z 113,A 136.8745,B 24.9326,C -1.8962,E1 24.875,E2 308.8305} C_DIS
LIN {X -82.7106,Y 68.7436,Z 113,A 135.374,B 24.9323,C -1.9003,E1 24.8776,E2 310.3284} C_DIS
LIN {X -80.6971,Y 71.098,Z 113,A 133.7424,B 24.932,C -1.9052,E1 24.8806,E2 311.9557} C_DIS
LIN {X -78.4545,Y 73.5639,Z 113,A 131.9196,B 24.9318,C -1.9079,E1 24.884,E2 313.78} C_DIS
LIN {X -76.171,Y 75.9273,Z 113,A 130.0236,B 24.9318,C -1.9068,E1 24.8878,E2 315.6867} C_DIS
LIN {X -73.6773,Y 78.3479,Z 113,A 128.3073,B 24.9312,C -1.9163,E1 24.8912,E2 317.3877} C_DIS
LIN {X -71.3922,Y 80.4369,Z 113,A 126.4985,B 24.9313,C -1.9141,E1 24.895,E2 319.2088} C_DIS
LIN {X -68.7256,Y 82.7256,Z 113,A 124.8087,B 24.9305,C -1.9251,E1 24.8985,E2 320.8788} C_DIS
LIN {X -66.6801,Y 84.383,Z 113,A 123.3405,B 24.9305,C -1.9257,E1 24.9018,E2 322.3511} C_DIS
LIN {X -64.068,Y 86.3855,Z 113,A 121.6373,B 24.9301,C -1.9313,E1 24.9055,E2 324.0473} C_DIS
LIN {X -61.9352,Y 87.9271,Z 113,A 120.2309,B 24.9299,C -1.934,E1 24.9087,E2 325.4521} C_DIS
LIN {X -58.9623,Y 89.9459,Z 113,A 118.2632,B 24.9297,C -1.9358,E1 24.9133,E2 327.4221} C_DIS
LIN {X -56.463,Y 91.5371,Z 113,A 116.7199,B 24.9294,C -1.94,E1 24.9169,E2 328.9601} C_DIS
LIN {X -53.3465,Y 93.386,Z 113,A 114.7836,B 24.9292,C -1.9433,E1 24.9216,E2 330.8944} C_DIS
LIN {X -50.707,Y 94.847,Z 113,A 113.1718,B 24.929,C -1.9459,E1 24.9255,E2 332.5047} C_DIS
LIN {X -47.5279,Y 96.4774,Z 113,A 111.2214,B 24.929,C -1.9473,E1 24.9304,E2 334.4571} C_DIS
LIN {X -45.1142,Y 97.6295,Z 113,A 109.8302,B 24.9287,C -1.9507,E1 24.9339,E2 335.8435} C_DIS
LIN {X -42.7101,Y 98.7049,Z 113,A 108.4227,B 24.9285,C -1.9527,E1 24.9375,E2 337.2498} C_DIS
LIN {X -40.2818,Y 99.7205,Z 113,A 106.9734,B 24.9285,C -1.9528,E1 24.9413,E2 338.7019} C_DIS
LIN {X -37.4717,Y 100.8119,Z 113,A 105.4054,B 24.9282,C -1.9564,E1 24.9453,E2 340.2647} C_DIS
LIN {X -34.9714,Y 101.7062,Z 113,A 103.9948,B 24.9281,C -1.9583,E1 24.949,E2 341.6734} C_DIS
LIN {X -32.4974,Y 102.5235,Z 113,A 102.5701,B 24.9281,C -1.9586,E1 24.9528,E2 343.1002} C_DIS
LIN {X -29.9165,Y 103.3059,Z 113,A 101.1742,B 24.9278,C -1.9617,E1 24.9566,E2 344.4909} C_DIS
LIN {X -27.393,Y 104.0037,Z 113,A 99.7657,B 24.9278,C -1.9627,E1 24.9604,E2 345.8994} C_DIS
LIN {X -23.9449,Y 104.8496,Z 113,A 97.6804,B 24.9282,C -1.957,E1 24.9661,E2 348.001} C_DIS
LIN {X -20.3445,Y 105.607,Z 113,A 95.8384,B 24.9277,C -1.9632,E1 24.9711,E2 349.8303} C_DIS
LIN {X -17.4616,Y 106.1221,Z 113,A 94.1487,B 24.928,C -1.9593,E1 24.9758,E2 351.5309} C_DIS
LIN {X -13.8627,Y 106.6516,Z 113,A 92.3251,B 24.9276,C -1.965,E1 24.9808,E2 353.3424} C_DIS
LIN {X -10.5329,Y 107.0337,Z 113,A 90.6107,B 24.9273,C -1.9687,E1 24.9855,E2 355.0491} C_DIS
LIN {X -7.9076,Y 107.2596,Z 113,A 89.2035,B 24.9273,C -1.9692,E1 24.9894,E2 356.4557} C_DIS
LIN {X -5.2789,Y 107.4211,Z 113,A 87.797,B 24.9273,C -1.9696,E1 24.9933,E2 357.8617} C_DIS
LIN {X -2.0702,Y 107.5288,Z 113,A 86.0214,B 24.9274,C -1.9675,E1 24.9983,E2 359.6424} C_DIS
LIN {X 1.3283,Y 107.5425,Z 113,A 84.2756,B 24.9272,C -1.9704,E1 25.0032,E2 361.3812} C_DIS
LIN {X 3.5798,Y 107.4895,Z 113,A 83.0327,B 24.9273,C -1.9688,E1 25.0066,E2 362.6276} C_DIS
LIN {X 6.2117,Y 107.3696,Z 113,A 81.6287,B 24.9273,C -1.9688,E1 25.0106,E2 364.0311} C_DIS
LIN {X 9.8445,Y 107.0972,Z 113,A 79.6845,B 24.9273,C -1.9686,E1 25.016,E2 365.9749} C_DIS
LIN {X 13.1728,Y 106.741,Z 113,A 77.9498,B 24.9273,C -1.9702,E1 25.0208,E2 367.7045} C_DIS
LIN {X 16.7074,Y 106.2435,Z 113,A 76.0052,B 24.9273,C -1.968,E1 25.0261,E2 369.6527} C_DIS
LIN {X 19.6811,Y 105.7346,Z 113,A 74.4417,B 24.9273,C -1.9691,E1 25.0304,E2 371.2117} C_DIS
LIN {X 23.2243,Y 105.0117,Z 113,A 72.472,B 24.9275,C -1.9665,E1 25.0358,E2 373.1852} C_DIS
LIN {X 26.141,Y 104.3255,Z 113,A 70.926,B 24.9275,C -1.9676,E1 25.04,E2 374.7264} C_DIS
LIN {X 28.3291,Y 103.751,Z 113,A 69.6751,B 24.9276,C -1.965,E1 25.0434,E2 375.9815} C_DIS
LIN {X 32.1172,Y 102.6416,Z 113,A 67.6194,B 24.9276,C -1.9653,E1 25.0489,E2 378.0328} C_DIS
LIN {X 34.9811,Y 101.7029,Z 113,A 66.0174,B 24.9276,C -1.9641,E1 25.0531,E2 379.6346} C_DIS
LIN {X 37.4791,Y 100.8091,Z 113,A 64.6087,B 24.9278,C -1.963,E1 25.0568,E2 381.0429} C_DIS
LIN {X 41.1586,Y 99.3636,Z 113,A 62.5045,B 24.9279,C -1.9609,E1 25.0623,E2 383.1473} C_DIS
LIN {X 43.9577,Y 98.1555,Z 113,A 60.789,B 24.9283,C -1.9554,E1 25.0667,E2 384.8718} C_DIS
LIN {X 46.8372,Y 96.8147,Z 113,A 59.1962,B 24.9282,C -1.9574,E1 25.0707,E2 386.4557} C_DIS
LIN {X 49.527,Y 95.4685,Z 113,A 57.5986,B 24.9283,C -1.9555,E1 25.0747,E2 388.0534} C_DIS
LIN {X 51.5307,Y 94.4002,Z 113,A 56.3491,B 24.9285,C -1.9522,E1 25.0777,E2 389.307} C_DIS
LIN {X 54.1588,Y 92.9192,Z 113,A 54.7909,B 24.9285,C -1.9519,E1 25.0815,E2 390.8613} C_DIS
LIN {X 57.2925,Y 91.0189,Z 113,A 52.8463,B 24.9288,C -1.9493,E1 25.0861,E2 392.8059} C_DIS
LIN {X 59.7859,Y 89.4022,Z 113,A 51.2732,B 24.9289,C -1.9471,E1 25.0898,E2 394.379} C_DIS
LIN {X 62.6933,Y 87.3863,Z 113,A 49.348,B 24.9293,C -1.9423,E1 25.0942,E2 396.3091} C_DIS
LIN {X 65.6475,Y 85.1888,Z 113,A 47.394,B 24.9295,C -1.9391,E1 25.0986,E2 398.2636} C_DIS
LIN {X 68.078,Y 83.2606,Z 113,A 45.6908,B 24.9299,C -1.9338,E1 25.1023,E2 399.9727} C_DIS
LIN {X 70.7388,Y 81.0108,Z 113,A 43.8945,B 24.9299,C -1.9327,E1 25.1061,E2 401.7646} C_DIS
LIN {X 73.0632,Y 78.9222,Z 113,A 42.2819,B 24.9301,C -1.9315,E1 25.1094,E2 403.3735} C_DIS
LIN {X 75.4444,Y 76.6479,Z 113,A 40.4838,B 24.9305,C -1.926,E1 25.113,E2 405.1772} C_DIS
LIN {X 77.5648,Y 74.5015,Z 113,A 38.876,B 24.9307,C -1.9225,E1 25.1162,E2 406.7864} C_DIS
LIN {X 79.9943,Y 71.8866,Z 113,A 36.9875,B 24.931,C -1.9187,E1 25.1197,E2 408.6754} C_DIS
LIN {X 81.9934,Y 69.5978,Z 113,A 35.3867,B 24.9312,C -1.9157,E1 25.1226,E2 410.276} C_DIS
LIN {X 84.2795,Y 66.8111,Z 113,A 33.4752,B 24.9315,C -1.9115,E1 25.126,E2 412.1886} C_DIS
LIN {X 86.1846,Y 64.3355,Z 113,A 31.8738,B 24.9316,C -1.9101,E1 25.1287,E2 413.7858} C_DIS
LIN {X 87.9361,Y 61.9225,Z 113,A 30.2878,B 24.9319,C -1.9062,E1 25.1313,E2 415.3733} C_DIS
LIN {X 89.9412,Y 58.9694,Z 113,A 28.3541,B 24.9323,C -1.8999,E1 25.1343,E2 417.3122} C_DIS
LIN {X 92.2478,Y 55.2947,Z 113,A 26.0976,B 24.9326,C -1.8961,E1 25.1376,E2 419.5662} C_DIS
LIN {X 93.3975,Y 53.3266,Z 113,A 24.8909,B 24.9328,C -1.8932,E1 25.1393,E2 420.7735} C_DIS
LIN {X 94.8533,Y 50.6953,Z 113,A 23.2995,B 24.9331,C -1.8892,E1 25.1414,E2 422.366} C_DIS
LIN {X 96.4771,Y 47.5287,Z 113,A 21.3675,B 24.9336,C -1.8824,E1 25.1439,E2 424.3039} C_DIS
LIN {X 98.1662,Y 43.9341,Z 113,A 19.3102,B 24.9338,C -1.8788,E1 25.1463,E2 426.3584} C_DIS
LIN {X 99.2129,Y 41.5164,Z 113,A 17.9259,B 24.9341,C -1.8756,E1 25.1478,E2 427.7427} C_DIS
LIN {X 100.3491,Y 38.6938,Z 113,A 16.3065,B 24.9344,C -1.8709,E1 25.1495,E2 429.3644} C_DIS
LIN {X 101.1047,Y 36.6689,Z 113,A 15.101,B 24.9348,C -1.8651,E1 25.1506,E2 430.5766} C_DIS
LIN {X 101.9998,Y 34.1004,Z 113,A 13.7047,B 24.9349,C -1.8631,E1 25.1519,E2 431.9699} C_DIS
LIN {X 102.9261,Y 31.1988,Z 113,A 12.1142,B 24.9352,C -1.8595,E1 25.1532,E2 433.5598} C_DIS
LIN {X 103.551,Y 29.0515,Z 113,A 10.8848,B 24.9355,C -1.8542,E1 25.1541,E2 434.7945} C_DIS
LIN {X 104.5415,Y 25.2558,Z 113,A 8.8449,B 24.9358,C -1.8499,E1 25.1556,E2 436.8329} C_DIS
LIN {X 105.1067,Y 22.7889,Z 113,A 7.435,B 24.9363,C -1.8431,E1 25.1564,E2 438.2507} C_DIS
LIN {X 105.7342,Y 19.6837,Z 113,A 5.8344,B 24.9364,C -1.8415,E1 25.1573,E2 439.8456} C_DIS
LIN {X 106.3859,Y 15.786,Z 113,A 3.7424,B 24.9369,C -1.8354,E1 25.1582,E2 441.9398} C_DIS
LIN {X 106.7753,Y 12.88,Z 113,A 2.0812,B 24.9375,C -1.8261,E1 25.1588,E2 443.613} C_DIS
LIN {X 107.1192,Y 9.6065,Z 113,A 0.4084,B 24.9376,C -1.824,E1 25.1592,E2 445.2809} C_DIS
LIN {X 107.3224,Y 6.9798,Z 113,A -0.9859,B 24.9379,C -1.8199,E1 25.1595,E2 446.6767} C_DIS
LIN {X 107.4611,Y 4.3489,Z 113,A -2.4989,B 24.9386,C -1.8106,E1 25.1597,E2 448.2025} C_DIS
LIN {X 107.548,Y 0.5646,Z 113,A -4.4441,B 24.9388,C -1.8072,E1 25.1597,E2 450.1443} C_DIS
LIN {X 107.5183,Y -2.6411,Z 113,A -6.0366,B 24.9388,C -1.8066,E1 25.1597,E2 451.7286} C_DIS
LIN {X 107.4297,Y -5.0788,Z 113,A -7.3111,B 24.939,C -1.8035,E1 25.1596,E2 453.0029} C_DIS
LIN {X 107.2599,Y -7.9035,Z 113,A -8.8227,B 24.9394,C -1.7984,E1 25.1593,E2 454.5175} C_DIS
LIN {X 107.0325,Y -10.5451,Z 113,A -10.2253,B 24.9397,C -1.7942,E1 25.1589,E2 455.9217} C_DIS
LIN {X 106.6215,Y -14.0951,Z 113,A -12.1762,B 24.9402,C -1.786,E1 25.1583,E2 457.8804} C_DIS
LIN {X 106.1807,Y -17.1111,Z 113,A -13.9037,B 24.9409,C -1.7762,E1 25.1575,E2 459.6208} C_DIS
LIN {X 105.5428,Y -20.6776,Z 113,A -15.6157,B 24.9406,C -1.7795,E1 25.1567,E2 461.3151} C_DIS
LIN {X 105.0212,Y -23.181,Z 113,A -17.0596,B 24.9412,C -1.7716,E1 25.1558,E2 462.7693} C_DIS
LIN {X 104.3214,Y -26.1567,Z 113,A -18.6118,B 24.9413,C -1.7697,E1 25.1548,E2 464.3171} C_DIS
LIN {X 103.753,Y -28.3216,Z 113,A -19.823,B 24.9416,C -1.7651,E1 25.1539,E2 465.5321} C_DIS
LIN {X 103.0234,Y -30.8707,Z 113,A -21.2036,B 24.9418,C -1.762,E1 25.1528,E2 466.9121} C_DIS
LIN {X 102.2381,Y -33.3792,Z 113,A -22.5619,B 24.942,C -1.7594,E1 25.1517,E2 468.2689} C_DIS
LIN {X 101.3917,Y -35.8683,Z 113,A -24.0278,B 24.9425,C -1.7521,E1 25.1503,E2 469.7435} C_DIS
LIN {X 100.0087,Y -39.5608,Z 113,A -26.1162,B 24.9429,C -1.7461,E1 25.1482,E2 471.8344} C_DIS
LIN {X 98.8511,Y -42.3749,Z 113,A -27.8261,B 24.9434,C -1.7373,E1 25.1464,E2 473.5559} C_DIS
LIN {X 97.491,Y -45.4118,Z 113,A -29.493,B 24.9434,C -1.7365,E1 25.1445,E2 475.2156} C_DIS
LIN {X 96.0598,Y -48.3701,Z 113,A -31.1821,B 24.9437,C -1.7338,E1 25.1424,E2 476.9019} C_DIS
LIN {X 94.8475,Y -50.7061,Z 113,A -32.5732,B 24.9439,C -1.7301,E1 25.1406,E2 478.2944} C_DIS
LIN {X 93.5782,Y -53.012,Z 113,A -34.153,B 24.9447,C -1.7183,E1 25.1384,E2 479.8938} C_DIS
LIN {X 91.71,Y -56.1797,Z 113,A -35.9149,B 24.9445,C -1.7212,E1 25.1359,E2 481.6399} C_DIS
LIN {X 90.3286,Y -58.3746,Z 113,A -37.3376,B 24.9448,C -1.7155,E1 25.1337,E2 483.069} C_DIS
LIN {X 88.6735,Y -60.8618,Z 113,A -38.8629,B 24.945,C -1.7138,E1 25.1313,E2 484.5906} C_DIS
LIN {X 86.3953,Y -64.0547,Z 113,A -40.9467,B 24.9453,C -1.7083,E1 25.1279,E2 486.6773} C_DIS
LIN {X 84.2884,Y -66.7998,Z 113,A -42.8448,B 24.9458,C -1.701,E1 25.1247,E2 488.5837} C_DIS
LIN {X 81.9915,Y -69.6,Z 113,A -44.7532,B 24.946,C -1.6968,E1 25.1213,E2 490.4932} C_DIS
LIN {X 80.1057,Y -71.7621,Z 113,A -46.2969,B 24.9463,C -1.6922,E1 25.1184,E2 492.0409} C_DIS
LIN {X 78.0199,Y -74.026,Z 113,A -48.0343,B 24.9469,C -1.6839,E1 25.1151,E2 493.7904} C_DIS
LIN {X 75.5801,Y -76.5139,Z 113,A -49.7391,B 24.9467,C -1.6858,E1 25.1117,E2 495.4833} C_DIS
LIN {X 73.2034,Y -78.7935,Z 113,A -51.5623,B 24.9472,C -1.6787,E1 25.108,E2 497.316} C_DIS
LIN {X 70.5715,Y -81.157,Z 113,A -53.3374,B 24.9472,C -1.679,E1 25.1043,E2 499.0832} C_DIS
LIN {X 68.0036,Y -83.3209,Z 113,A -55.2214,B 24.9477,C -1.6709,E1 25.1002,E2 500.9791} C_DIS
LIN {X 65.2434,Y -85.5002,Z 113,A -56.9822,B 24.9477,C -1.6716,E1 25.0964,E2 502.7318} C_DIS
LIN {X 63.3042,Y -86.9447,Z 113,A -58.2862,B 24.9478,C -1.6682,E1 25.0934,E2 504.0391} C_DIS
LIN {X 60.8212,Y -88.7012,Z 113,A -59.8466,B 24.9478,C -1.6674,E1 25.0899,E2 505.596} C_DIS
LIN {X 57.5254,Y -90.8734,Z 113,A -61.9523,B 24.9482,C -1.6632,E1 25.0849,E2 507.7048} C_DIS
LIN {X 55.2854,Y -92.2533,Z 113,A -63.3465,B 24.9483,C -1.6609,E1 25.0816,E2 509.1002} C_DIS
LIN {X 52.1966,Y -94.0336,Z 113,A -65.284,B 24.9486,C -1.6559,E1 25.0769,E2 511.0438} C_DIS
LIN {X 48.9881,Y -95.7439,Z 113,A -67.2415,B 24.9489,C -1.6517,E1 25.072,E2 513.0056} C_DIS
LIN {X 45.9817,Y -97.2257,Z 113,A -68.9504,B 24.9489,C -1.652,E1 25.0677,E2 514.7093} C_DIS
LIN {X 42.683,Y -98.7167,Z 113,A -70.8734,B 24.949,C -1.6493,E1 25.0628,E2 516.634} C_DIS
LIN {X 40.2605,Y -99.7292,Z 113,A -72.2818,B 24.9492,C -1.6468,E1 25.0592,E2 518.0449} C_DIS
LIN {X 37.4592,Y -100.8164,Z 113,A -73.8576,B 24.9492,C -1.6457,E1 25.0551,E2 519.62} C_DIS
LIN {X 34.9865,Y -101.7011,Z 113,A -75.2591,B 24.9494,C -1.6438,E1 25.0514,E2 521.0232} C_DIS
LIN {X 32.423,Y -102.5468,Z 113,A -76.6835,B 24.9494,C -1.6426,E1 25.0476,E2 522.4477} C_DIS
LIN {X 29.9368,Y -103.3002,Z 113,A -78.0653,B 24.9495,C -1.6411,E1 25.0439,E2 523.8307} C_DIS
LIN {X 27.429,Y -103.9942,Z 113,A -79.4537,B 24.9496,C -1.6395,E1 25.0402,E2 525.2206} C_DIS
LIN {X 24.0163,Y -104.8331,Z 113,A -81.3693,B 24.9499,C -1.6359,E1 25.0349,E2 527.142} C_DIS
LIN {X 20.9684,Y -105.4868,Z 113,A -82.9819,B 24.9499,C -1.6364,E1 25.0305,E2 528.7514} C_DIS
LIN {X 17.4566,Y -106.1229,Z 113,A -84.9237,B 24.95,C -1.6332,E1 25.0252,E2 530.6985} C_DIS
LIN {X 14.4735,Y -106.5724,Z 113,A -86.4859,B 24.95,C -1.6339,E1 25.0209,E2 532.2578} C_DIS
LIN {X 11.1806,Y -106.966,Z 113,A -88.3024,B 24.9502,C -1.6309,E1 25.0158,E2 534.0802} C_DIS
LIN {X 8.0834,Y -107.2456,Z 113,A -89.8906,B 24.95,C -1.6328,E1 25.0114,E2 535.6629} C_DIS
LIN {X 5.2717,Y -107.4214,Z 113,A -91.4027,B 24.9501,C -1.6317,E1 25.0072,E2 537.177} C_DIS
LIN {X 2.6394,Y -107.5184,Z 113,A -92.8076,B 24.9501,C -1.6312,E1 25.0033,E2 538.5829} C_DIS
LIN {X 2.6394,Y -107.5184,Z 113,A -92.8076,B 24.9501,C -1.6312,E1 25.0033,E2 538.5829} C_DIS
Enddeposition()
LIN {X 0.7991,Y -113.7938,Z 114,A -93.153,B 24.9546,C -1.5563,E1 25.0018,E2 539.1057} C_DIS
Startdeposition()
$VEL.CP = VEL_PRINT
LIN {X 3.1462,Y -113.7549,Z 114,A -91.7689,B 24.9541,C -1.5655,E1 25.0057,E2 537.7001} C_DIS
LIN {X 5.5839,Y -113.663,Z 114,A -90.4389,B 24.9538,C -1.5704,E1 25.0095,E2 536.3589} C_DIS
LIN {X 8.7285,Y -113.4632,Z 114,A -88.9583,B 24.954,C -1.5665,E1 25.0136,E2 534.8882} C_DIS
LIN {X 11.5104,Y -113.2148,Z 114,A -87.6952,B 24.9543,C -1.561,E1 25.017,E2 533.639} C_DIS
LIN {X 14.2853,Y -112.8982,Z 114,A -86.149,B 24.9539,C -1.568,E1 25.0214,E2 532.0773} C_DIS
LIN {X 17.0517,Y -112.5136,Z 114,A -84.7451,B 24.9539,C -1.5689,E1 25.0253,E2 530.6726} C_DIS
LIN {X 19.4555,Y -112.1246,Z 114,A -83.521,B 24.9539,C -1.5697,E1 25.0286,E2 529.4478} C_DIS
LIN {X 22.5519,Y -111.5414,Z 114,A -82.1006,B 24.9542,C -1.5637,E1 25.0325,E2 528.0433} C_DIS
LIN {X 24.9337,Y -111.0349,Z 114,A -80.7139,B 24.9537,C -1.572,E1 25.0363,E2 526.6388} C_DIS
LIN {X 27.9979,Y -110.3005,Z 114,A -79.1309,B 24.9537,C -1.5734,E1 25.0406,E2 525.0547} C_DIS
LIN {X 30.6963,Y -109.5802,Z 114,A -77.7279,B 24.9535,C -1.5748,E1 25.0444,E2 523.6508} C_DIS
LIN {X 33.0344,Y -108.8999,Z 114,A -76.5049,B 24.9535,C -1.576,E1 25.0477,E2 522.4269} C_DIS
LIN {X 35.697,Y -108.0564,Z 114,A -75.1024,B 24.9534,C -1.5776,E1 25.0514,E2 521.0234} C_DIS
LIN {X 38.3381,Y -107.1478,Z 114,A -73.6999,B 24.9533,C -1.5793,E1 25.0551,E2 519.6197} C_DIS
LIN {X 41.2893,Y -106.0437,Z 114,A -72.1183,B 24.9532,C -1.5812,E1 25.0592,E2 518.0369} C_DIS
LIN {X 43.8793,Y -104.9985,Z 114,A -70.7163,B 24.953,C -1.5831,E1 25.0628,E2 516.6337} C_DIS
LIN {X 46.4428,Y -103.89,Z 114,A -69.3146,B 24.953,C -1.585,E1 25.0664,E2 515.2308} C_DIS
LIN {X 48.6558,Y -102.874,Z 114,A -67.9632,B 24.9525,C -1.5926,E1 25.0699,E2 513.865} C_DIS
LIN {X 51.4845,Y -101.4861,Z 114,A -66.512,B 24.9527,C -1.5892,E1 25.0735,E2 512.4259} C_DIS
LIN {X 53.9596,Y -100.192,Z 114,A -65.1108,B 24.9525,C -1.5914,E1 25.0769,E2 511.0234} C_DIS
LIN {X 56.0918,Y -99.0159,Z 114,A -63.8895,B 24.9525,C -1.5933,E1 25.0799,E2 509.8012} C_DIS
LIN {X 58.8108,Y -97.4236,Z 114,A -62.3094,B 24.9523,C -1.596,E1 25.0837,E2 508.2196} C_DIS
LIN {X 61.184,Y -95.951,Z 114,A -61.072,B 24.9526,C -1.591,E1 25.0866,E2 506.9979} C_DIS
LIN {X 63.2239,Y -94.6213,Z 114,A -59.5586,B 24.9516,C -1.6066,E1 25.0902,E2 505.4528} C_DIS
LIN {X 65.8184,Y -92.8333,Z 114,A -58.2713,B 24.9523,C -1.5961,E1 25.0931,E2 504.1945} C_DIS
LIN {X 68.0768,Y -91.19,Z 114,A -56.8713,B 24.9521,C -1.5988,E1 25.0962,E2 502.7932} C_DIS
LIN {X 70.2942,Y -89.4919,Z 114,A -55.4715,B 24.9519,C -1.6016,E1 25.0993,E2 501.392} C_DIS
LIN {X 72.194,Y -87.9686,Z 114,A -53.9595,B 24.951,C -1.6174,E1 25.1027,E2 499.8483} C_DIS
LIN {X 74.3311,Y -86.1704,Z 114,A -52.56,B 24.9508,C -1.6203,E1 25.1056,E2 498.4475} C_DIS
LIN {X 76.6872,Y -84.0782,Z 114,A -51.111,B 24.951,C -1.6177,E1 25.1086,E2 497.0104} C_DIS
LIN {X 78.7275,Y -82.1709,Z 114,A -49.7118,B 24.9508,C -1.6208,E1 25.1115,E2 495.6097} C_DIS
LIN {X 80.4688,Y -80.4688,Z 114,A -48.492,B 24.9506,C -1.6235,E1 25.1139,E2 494.3887} C_DIS
LIN {X 82.4194,Y -78.4697,Z 114,A -47.0935,B 24.9504,C -1.6266,E1 25.1166,E2 492.9887} C_DIS
LIN {X 84.3203,Y -76.4234,Z 114,A -45.5656,B 24.9499,C -1.6359,E1 25.1195,E2 491.4459} C_DIS
LIN {X 86.1704,Y -74.3311,Z 114,A -44.161,B 24.9496,C -1.6395,E1 25.1221,E2 490.0392} C_DIS
LIN {X 88.194,Y -71.9159,Z 114,A -42.8814,B 24.9502,C -1.6295,E1 25.1243,E2 488.7891} C_DIS
LIN {X 89.9324,Y -69.7298,Z 114,A -41.4834,B 24.95,C -1.6329,E1 25.1267,E2 487.3895} C_DIS
LIN {X 91.6165,Y -67.5018,Z 114,A -40.0853,B 24.9498,C -1.6363,E1 25.1291,E2 485.99} C_DIS
LIN {X 93.0412,Y -65.527,Z 114,A -38.5748,B 24.9488,C -1.6529,E1 25.1316,E2 484.4476} C_DIS
LIN {X 94.8183,Y -62.9251,Z 114,A -37.2897,B 24.9494,C -1.6434,E1 25.1335,E2 483.1913} C_DIS
LIN {X 96.1444,Y -60.8828,Z 114,A -35.9088,B 24.9487,C -1.6541,E1 25.1356,E2 481.7922} C_DIS
LIN {X 97.7917,Y -58.1967,Z 114,A -34.332,B 24.9485,C -1.6583,E1 25.1379,E2 480.2135} C_DIS
LIN {X 99.6968,Y -54.8725,Z 114,A -32.4148,B 24.9482,C -1.6634,E1 25.1406,E2 478.2943} C_DIS
LIN {X 101.0134,Y -52.4093,Z 114,A -31.0177,B 24.9479,C -1.6671,E1 25.1424,E2 476.8957} C_DIS
LIN {X 102.4242,Y -49.5919,Z 114,A -29.6037,B 24.9481,C -1.6639,E1 25.1441,E2 475.4969} C_DIS
LIN {X 103.4634,Y -47.3897,Z 114,A -28.2234,B 24.9474,C -1.6748,E1 25.1458,E2 474.0983} C_DIS
LIN {X 104.5952,Y -44.8363,Z 114,A -26.8263,B 24.9472,C -1.6787,E1 25.1473,E2 472.6997} C_DIS
LIN {X 105.664,Y -42.2559,Z 114,A -25.3003,B 24.9466,C -1.6887,E1 25.1489,E2 471.1586} C_DIS
LIN {X 106.7919,Y -39.3138,Z 114,A -23.8537,B 24.9466,C -1.6871,E1 25.1503,E2 469.7237} C_DIS
LIN {X 107.7245,Y -36.6811,Z 114,A -22.4567,B 24.9464,C -1.6911,E1 25.1516,E2 468.3252} C_DIS
LIN {X 108.5923,Y -34.0264,Z 114,A -21.2222,B 24.9466,C -1.6875,E1 25.1527,E2 467.1061} C_DIS
LIN {X 109.297,Y -31.6956,Z 114,A -19.8422,B 24.9459,C -1.6986,E1 25.1538,E2 465.7079} C_DIS
LIN {X 110.042,Y -29.0037,Z 114,A -18.3165,B 24.9453,C -1.7087,E1 25.1549,E2 464.1671} C_DIS
LIN {X 110.8012,Y -25.9456,Z 114,A -16.8701,B 24.9453,C -1.7073,E1 25.1558,E2 462.7325} C_DIS
LIN {X 111.3326,Y -23.5693,Z 114,A -15.5233,B 24.9448,C -1.7168,E1 25.1566,E2 461.3709} C_DIS
LIN {X 111.9408,Y -20.4776,Z 114,A -14.2392,B 24.9453,C -1.7078,E1 25.1573,E2 460.1156} C_DIS
LIN {X 112.3549,Y -18.0781,Z 114,A -12.8595,B 24.9446,C -1.719,E1 25.1579,E2 458.7178} C_DIS
LIN {X 112.7648,Y -15.3153,Z 114,A -11.3338,B 24.944,C -1.7292,E1 25.1585,E2 457.177} C_DIS
LIN {X 113.1067,Y -12.5433,Z 114,A -10.0664,B 24.944,C -1.7272,E1 25.1589,E2 455.9216} C_DIS
LIN {X 113.4088,Y -9.4092,Z 114,A -8.4912,B 24.9438,C -1.7319,E1 25.1593,E2 454.3447} C_DIS
LIN {X 113.6056,Y -6.6209,Z 114,A -7.2569,B 24.944,C -1.7284,E1 25.1595,E2 453.126} C_DIS
LIN {X 113.7339,Y -3.8309,Z 114,A -5.8603,B 24.9437,C -1.7326,E1 25.1597,E2 451.728} C_DIS
LIN {X 113.7915,Y -1.3965,Z 114,A -4.4731,B 24.943,C -1.7441,E1 25.1597,E2 450.3219} C_DIS
LIN {X 113.7849,Y 1.7544,Z 114,A -3.0674,B 24.9432,C -1.7408,E1 25.1597,E2 448.9323} C_DIS
LIN {X 113.7076,Y 4.5463,Z 114,A -1.6708,B 24.9429,C -1.7449,E1 25.1597,E2 447.5342} C_DIS
LIN {X 113.5617,Y 7.3355,Z 114,A -0.0364,B 24.9419,C -1.7601,E1 25.1594,E2 445.8737} C_DIS
LIN {X 113.3475,Y 10.1202,Z 114,A 1.2844,B 24.9419,C -1.7606,E1 25.1591,E2 444.5595} C_DIS
LIN {X 113.1067,Y 12.5433,Z 114,A 2.6313,B 24.9413,C -1.7702,E1 25.1587,E2 443.198} C_DIS
LIN {X 112.7648,Y 15.3153,Z 114,A 4.0282,B 24.941,C -1.7743,E1 25.1581,E2 441.7998} C_DIS
LIN {X 112.2959,Y 18.4311,Z 114,A 5.4746,B 24.941,C -1.7728,E1 25.1575,E2 440.3654} C_DIS
LIN {X 111.8774,Y 20.8299,Z 114,A 6.8215,B 24.9405,C -1.7823,E1 25.1568,E2 439.004} C_DIS
LIN {X 111.3326,Y 23.5693,Z 114,A 8.2183,B 24.9402,C -1.7862,E1 25.156,E2 437.606} C_DIS
LIN {X 110.7206,Y 26.2944,Z 114,A 9.6153,B 24.9399,C -1.7902,E1 25.1551,E2 436.2078} C_DIS
LIN {X 109.9486,Y 29.3493,Z 114,A 11.062,B 24.94,C -1.7886,E1 25.1541,E2 434.7731} C_DIS
LIN {X 109.1952,Y 32.0387,Z 114,A 12.4832,B 24.9397,C -1.7936,E1 25.153,E2 433.3483} C_DIS
LIN {X 108.4863,Y 34.3683,Z 114,A 13.832,B 24.9391,C -1.803,E1 25.1519,E2 431.9849} C_DIS
LIN {X 107.4015,Y 37.6149,Z 114,A 15.3056,B 24.9395,C -1.7966,E1 25.1506,E2 430.5347} C_DIS
LIN {X 106.5424,Y 39.9848,Z 114,A 16.6507,B 24.939,C -1.8039,E1 25.1493,E2 429.18} C_DIS
LIN {X 105.5291,Y 42.5875,Z 114,A 18.048,B 24.9388,C -1.8077,E1 25.1478,E2 427.7816} C_DIS
LIN {X 104.4521,Y 45.1645,Z 114,A 19.2831,B 24.939,C -1.8038,E1 25.1465,E2 426.5623} C_DIS
LIN {X 103.4634,Y 47.3897,Z 114,A 20.7935,B 24.9379,C -1.8205,E1 25.1447,E2 425.0208} C_DIS
LIN {X 102.1102,Y 50.2353,Z 114,A 22.241,B 24.938,C -1.8186,E1 25.143,E2 423.5856} C_DIS
LIN {X 101.0134,Y 52.4093,Z 114,A 23.5889,B 24.9374,C -1.8276,E1 25.1412,E2 422.2235} C_DIS
LIN {X 99.5223,Y 55.1851,Z 114,A 25.0369,B 24.9375,C -1.8256,E1 25.1393,E2 420.7878} C_DIS
LIN {X 98.138,Y 57.6109,Z 114,A 26.4352,B 24.9373,C -1.8291,E1 25.1374,E2 419.3886} C_DIS
LIN {X 96.6946,Y 60.0019,Z 114,A 27.8957,B 24.9369,C -1.8353,E1 25.1352,E2 417.9207} C_DIS
LIN {X 95.2483,Y 62.2729,Z 114,A 29.0643,B 24.9372,C -1.8303,E1 25.1335,E2 416.77} C_DIS
LIN {X 93.8383,Y 64.3803,Z 114,A 30.4509,B 24.9366,C -1.8386,E1 25.1313,E2 415.3706} C_DIS
LIN {X 92.2301,Y 66.6638,Z 114,A 31.979,B 24.936,C -1.8477,E1 25.1288,E2 413.8284} C_DIS
LIN {X 90.3478,Y 69.1907,Z 114,A 33.4275,B 24.9362,C -1.8453,E1 25.1264,E2 412.3923} C_DIS
LIN {X 88.7483,Y 71.232,Z 114,A 34.797,B 24.9357,C -1.8514,E1 25.124,E2 411.015} C_DIS
LIN {X 86.8439,Y 73.5405,Z 114,A 36.3117,B 24.9355,C -1.8553,E1 25.1212,E2 409.4979} C_DIS
LIN {X 84.3203,Y 76.4234,Z 114,A 38.1454,B 24.9355,C -1.8553,E1 25.1179,E2 407.6723} C_DIS
LIN {X 82.1709,Y 78.7275,Z 114,A 39.5613,B 24.9358,C -1.8512,E1 25.1152,E2 406.2725} C_DIS
LIN {X 80.4688,Y 80.4688,Z 114,A 41.0742,B 24.9347,C -1.8668,E1 25.1121,E2 404.729} C_DIS
LIN {X 78.209,Y 82.6646,Z 114,A 42.5238,B 24.9349,C -1.864,E1 25.1092,E2 403.2921} C_DIS
LIN {X 76.4234,Y 84.3203,Z 114,A 43.7444,B 24.9347,C -1.8662,E1 25.1067,E2 402.0713} C_DIS
LIN {X 74.0586,Y 86.4026,Z 114,A 45.1614,B 24.935,C -1.8617,E1 25.1038,E2 400.6703} C_DIS
LIN {X 72.194,Y 87.9686,Z 114,A 46.675,B 24.934,C -1.877,E1 25.1005,E2 399.1264} C_DIS
LIN {X 69.7298,Y 89.9324,Z 114,A 47.9625,B 24.9347,C -1.8665,E1 25.0977,E2 397.8685} C_DIS
LIN {X 67.5018,Y 91.6165,Z 114,A 49.5263,B 24.934,C -1.8761,E1 25.0942,E2 396.2877} C_DIS
LIN {X 65.2331,Y 93.2455,Z 114,A 50.9276,B 24.9339,C -1.8783,E1 25.091,E2 394.8861} C_DIS
LIN {X 62.9251,Y 94.8183,Z 114,A 52.1656,B 24.9342,C -1.8731,E1 25.0881,E2 393.6646} C_DIS
LIN {X 60.8828,Y 96.1444,Z 114,A 53.6355,B 24.9333,C -1.8859,E1 25.0846,E2 392.1691} C_DIS
LIN {X 58.5049,Y 97.6096,Z 114,A 54.9523,B 24.9335,C -1.884,E1 25.0815,E2 390.8608} C_DIS
LIN {X 55.7793,Y 99.1905,Z 114,A 56.5337,B 24.9333,C -1.8861,E1 25.0777,E2 389.2793} C_DIS
LIN {X 53.3282,Y 100.5295,Z 114,A 57.773,B 24.9337,C -1.8806,E1 25.0747,E2 388.0565} C_DIS
LIN {X 51.1658,Y 101.649,Z 114,A 59.2884,B 24.9327,C -1.895,E1 25.0708,E2 386.5112} C_DIS
LIN {X 48.3313,Y 103.0251,Z 114,A 60.7409,B 24.933,C -1.8911,E1 25.0672,E2 385.0719} C_DIS
Enddeposition()
END
